// TIA Portal V19 export
FUNCTION "AUTO_SUBOUTPUT" : Void   // FC11, LAD
{ S7_Optimized_Access := 'TRUE' }
// stored: SetENOAutomatically false
BEGIN

REGION Network 1: MGF FEED PUMP P-101 A
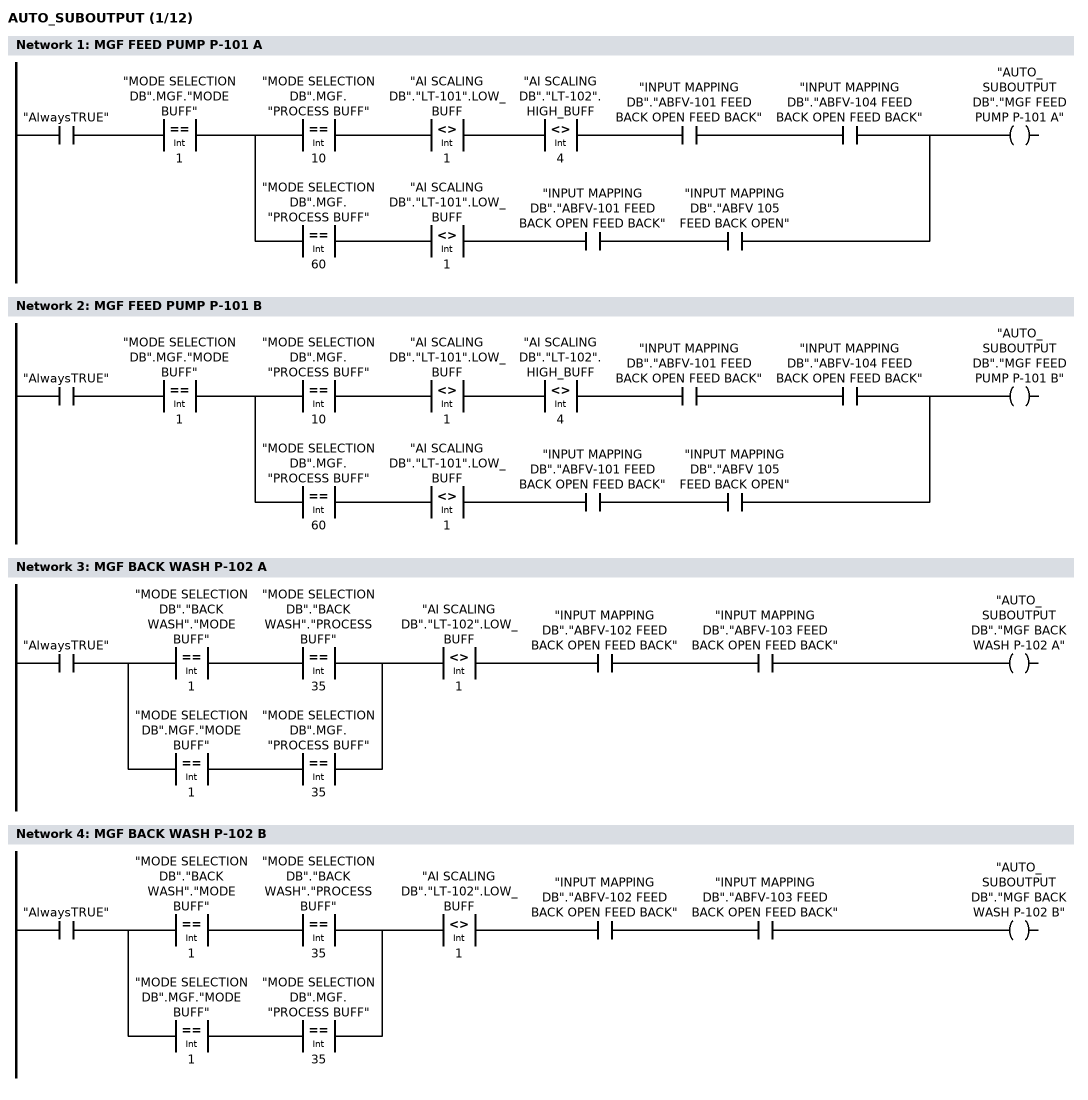
   RUNG wire#powerrail
      Contact( "AlwaysTRUE" )
      { S7_Templates := "SrcType := Int" } EQ_Contact(in1 := "MODE SELECTION DB".MGF."MODE BUFF", in2 := 1)
      wire#w1
      { S7_Templates := "SrcType := Int" } EQ_Contact(in1 := "MODE SELECTION DB".MGF."PROCESS BUFF", in2 := 10)
      { S7_Templates := "SrcType := Int" } NE_Contact(in1 := "AI SCALING DB"."LT-101".LOW_BUFF, in2 := 1)
      { S7_Templates := "SrcType := Int" } NE_Contact(in1 := "AI SCALING DB"."LT-102".HIGH_BUFF, in2 := 4)
      Contact( "INPUT MAPPING DB"."ABFV-101 FEED BACK OPEN FEED BACK" )
      Contact( "INPUT MAPPING DB"."ABFV-104 FEED BACK OPEN FEED BACK" )
      wire#w2
      Coil( "AUTO_SUBOUTPUT DB"."MGF FEED PUMP P-101 A" )
   END_RUNG
   RUNG wire#w1
      { S7_Templates := "SrcType := Int" } EQ_Contact(in1 := "MODE SELECTION DB".MGF."PROCESS BUFF", in2 := 60)
      { S7_Templates := "SrcType := Int" } NE_Contact(in1 := "AI SCALING DB"."LT-101".LOW_BUFF, in2 := 1)
      Contact( "INPUT MAPPING DB"."ABFV-101 FEED BACK OPEN FEED BACK" )
      Contact( "INPUT MAPPING DB"."ABFV 105 FEED BACK OPEN" )
   END_RUNG wire#w2
   // the same network as SCL:
   "AUTO_SUBOUTPUT DB"."MGF FEED PUMP P-101 A" := "AlwaysTRUE" AND ("MODE SELECTION DB".MGF."MODE BUFF" = 1) AND ((("MODE SELECTION DB".MGF."PROCESS BUFF" = 10) AND ("AI SCALING DB"."LT-101".LOW_BUFF <> 1) AND ("AI SCALING DB"."LT-102".HIGH_BUFF <> 4) AND "INPUT MAPPING DB"."ABFV-101 FEED BACK OPEN FEED BACK" AND "INPUT MAPPING DB"."ABFV-104 FEED BACK OPEN FEED BACK") OR (("MODE SELECTION DB".MGF."PROCESS BUFF" = 60) AND ("AI SCALING DB"."LT-101".LOW_BUFF <> 1) AND "INPUT MAPPING DB"."ABFV-101 FEED BACK OPEN FEED BACK" AND "INPUT MAPPING DB"."ABFV 105 FEED BACK OPEN"));
END_REGION

REGION Network 2: MGF FEED PUMP P-101 B
   RUNG wire#powerrail
      Contact( "AlwaysTRUE" )
      { S7_Templates := "SrcType := Int" } EQ_Contact(in1 := "MODE SELECTION DB".MGF."MODE BUFF", in2 := 1)
      wire#w1
      { S7_Templates := "SrcType := Int" } EQ_Contact(in1 := "MODE SELECTION DB".MGF."PROCESS BUFF", in2 := 10)
      { S7_Templates := "SrcType := Int" } NE_Contact(in1 := "AI SCALING DB"."LT-101".LOW_BUFF, in2 := 1)
      { S7_Templates := "SrcType := Int" } NE_Contact(in1 := "AI SCALING DB"."LT-102".HIGH_BUFF, in2 := 4)
      Contact( "INPUT MAPPING DB"."ABFV-101 FEED BACK OPEN FEED BACK" )
      Contact( "INPUT MAPPING DB"."ABFV-104 FEED BACK OPEN FEED BACK" )
      wire#w2
      Coil( "AUTO_SUBOUTPUT DB"."MGF FEED PUMP P-101 B" )
   END_RUNG
   RUNG wire#w1
      { S7_Templates := "SrcType := Int" } EQ_Contact(in1 := "MODE SELECTION DB".MGF."PROCESS BUFF", in2 := 60)
      { S7_Templates := "SrcType := Int" } NE_Contact(in1 := "AI SCALING DB"."LT-101".LOW_BUFF, in2 := 1)
      Contact( "INPUT MAPPING DB"."ABFV-101 FEED BACK OPEN FEED BACK" )
      Contact( "INPUT MAPPING DB"."ABFV 105 FEED BACK OPEN" )
   END_RUNG wire#w2
   // the same network as SCL:
   "AUTO_SUBOUTPUT DB"."MGF FEED PUMP P-101 B" := "AlwaysTRUE" AND ("MODE SELECTION DB".MGF."MODE BUFF" = 1) AND ((("MODE SELECTION DB".MGF."PROCESS BUFF" = 10) AND ("AI SCALING DB"."LT-101".LOW_BUFF <> 1) AND ("AI SCALING DB"."LT-102".HIGH_BUFF <> 4) AND "INPUT MAPPING DB"."ABFV-101 FEED BACK OPEN FEED BACK" AND "INPUT MAPPING DB"."ABFV-104 FEED BACK OPEN FEED BACK") OR (("MODE SELECTION DB".MGF."PROCESS BUFF" = 60) AND ("AI SCALING DB"."LT-101".LOW_BUFF <> 1) AND "INPUT MAPPING DB"."ABFV-101 FEED BACK OPEN FEED BACK" AND "INPUT MAPPING DB"."ABFV 105 FEED BACK OPEN"));
END_REGION

REGION Network 3: MGF BACK WASH P-102 A
   RUNG wire#powerrail
      Contact( "AlwaysTRUE" )
      wire#w1
      { S7_Templates := "SrcType := Int" } EQ_Contact(in1 := "MODE SELECTION DB"."BACK WASH"."MODE BUFF", in2 := 1)
      { S7_Templates := "SrcType := Int" } EQ_Contact(in1 := "MODE SELECTION DB"."BACK WASH"."PROCESS BUFF", in2 := 35)
      wire#w2
      { S7_Templates := "SrcType := Int" } NE_Contact(in1 := "AI SCALING DB"."LT-102".LOW_BUFF, in2 := 1)
      Contact( "INPUT MAPPING DB"."ABFV-102 FEED BACK OPEN FEED BACK" )
      Contact( "INPUT MAPPING DB"."ABFV-103 FEED BACK OPEN FEED BACK" )
      Coil( "AUTO_SUBOUTPUT DB"."MGF BACK WASH P-102 A" )
   END_RUNG
   RUNG wire#w1
      { S7_Templates := "SrcType := Int" } EQ_Contact(in1 := "MODE SELECTION DB".MGF."MODE BUFF", in2 := 1)
      { S7_Templates := "SrcType := Int" } EQ_Contact(in1 := "MODE SELECTION DB".MGF."PROCESS BUFF", in2 := 35)
   END_RUNG wire#w2
   // the same network as SCL:
   "AUTO_SUBOUTPUT DB"."MGF BACK WASH P-102 A" := "AlwaysTRUE" AND ((("MODE SELECTION DB"."BACK WASH"."MODE BUFF" = 1) AND ("MODE SELECTION DB"."BACK WASH"."PROCESS BUFF" = 35)) OR (("MODE SELECTION DB".MGF."MODE BUFF" = 1) AND ("MODE SELECTION DB".MGF."PROCESS BUFF" = 35))) AND ("AI SCALING DB"."LT-102".LOW_BUFF <> 1) AND "INPUT MAPPING DB"."ABFV-102 FEED BACK OPEN FEED BACK" AND "INPUT MAPPING DB"."ABFV-103 FEED BACK OPEN FEED BACK";
END_REGION

REGION Network 4: MGF BACK WASH P-102 B
   RUNG wire#powerrail
      Contact( "AlwaysTRUE" )
      wire#w1
      { S7_Templates := "SrcType := Int" } EQ_Contact(in1 := "MODE SELECTION DB"."BACK WASH"."MODE BUFF", in2 := 1)
      { S7_Templates := "SrcType := Int" } EQ_Contact(in1 := "MODE SELECTION DB"."BACK WASH"."PROCESS BUFF", in2 := 35)
      wire#w2
      { S7_Templates := "SrcType := Int" } NE_Contact(in1 := "AI SCALING DB"."LT-102".LOW_BUFF, in2 := 1)
      Contact( "INPUT MAPPING DB"."ABFV-102 FEED BACK OPEN FEED BACK" )
      Contact( "INPUT MAPPING DB"."ABFV-103 FEED BACK OPEN FEED BACK" )
      Coil( "AUTO_SUBOUTPUT DB"."MGF BACK WASH P-102 B" )
   END_RUNG
   RUNG wire#w1
      { S7_Templates := "SrcType := Int" } EQ_Contact(in1 := "MODE SELECTION DB".MGF."MODE BUFF", in2 := 1)
      { S7_Templates := "SrcType := Int" } EQ_Contact(in1 := "MODE SELECTION DB".MGF."PROCESS BUFF", in2 := 35)
   END_RUNG wire#w2
   // the same network as SCL:
   "AUTO_SUBOUTPUT DB"."MGF BACK WASH P-102 B" := "AlwaysTRUE" AND ((("MODE SELECTION DB"."BACK WASH"."MODE BUFF" = 1) AND ("MODE SELECTION DB"."BACK WASH"."PROCESS BUFF" = 35)) OR (("MODE SELECTION DB".MGF."MODE BUFF" = 1) AND ("MODE SELECTION DB".MGF."PROCESS BUFF" = 35))) AND ("AI SCALING DB"."LT-102".LOW_BUFF <> 1) AND "INPUT MAPPING DB"."ABFV-102 FEED BACK OPEN FEED BACK" AND "INPUT MAPPING DB"."ABFV-103 FEED BACK OPEN FEED BACK";
END_REGION

REGION Network 5: UF FEED PUMP P-103 A
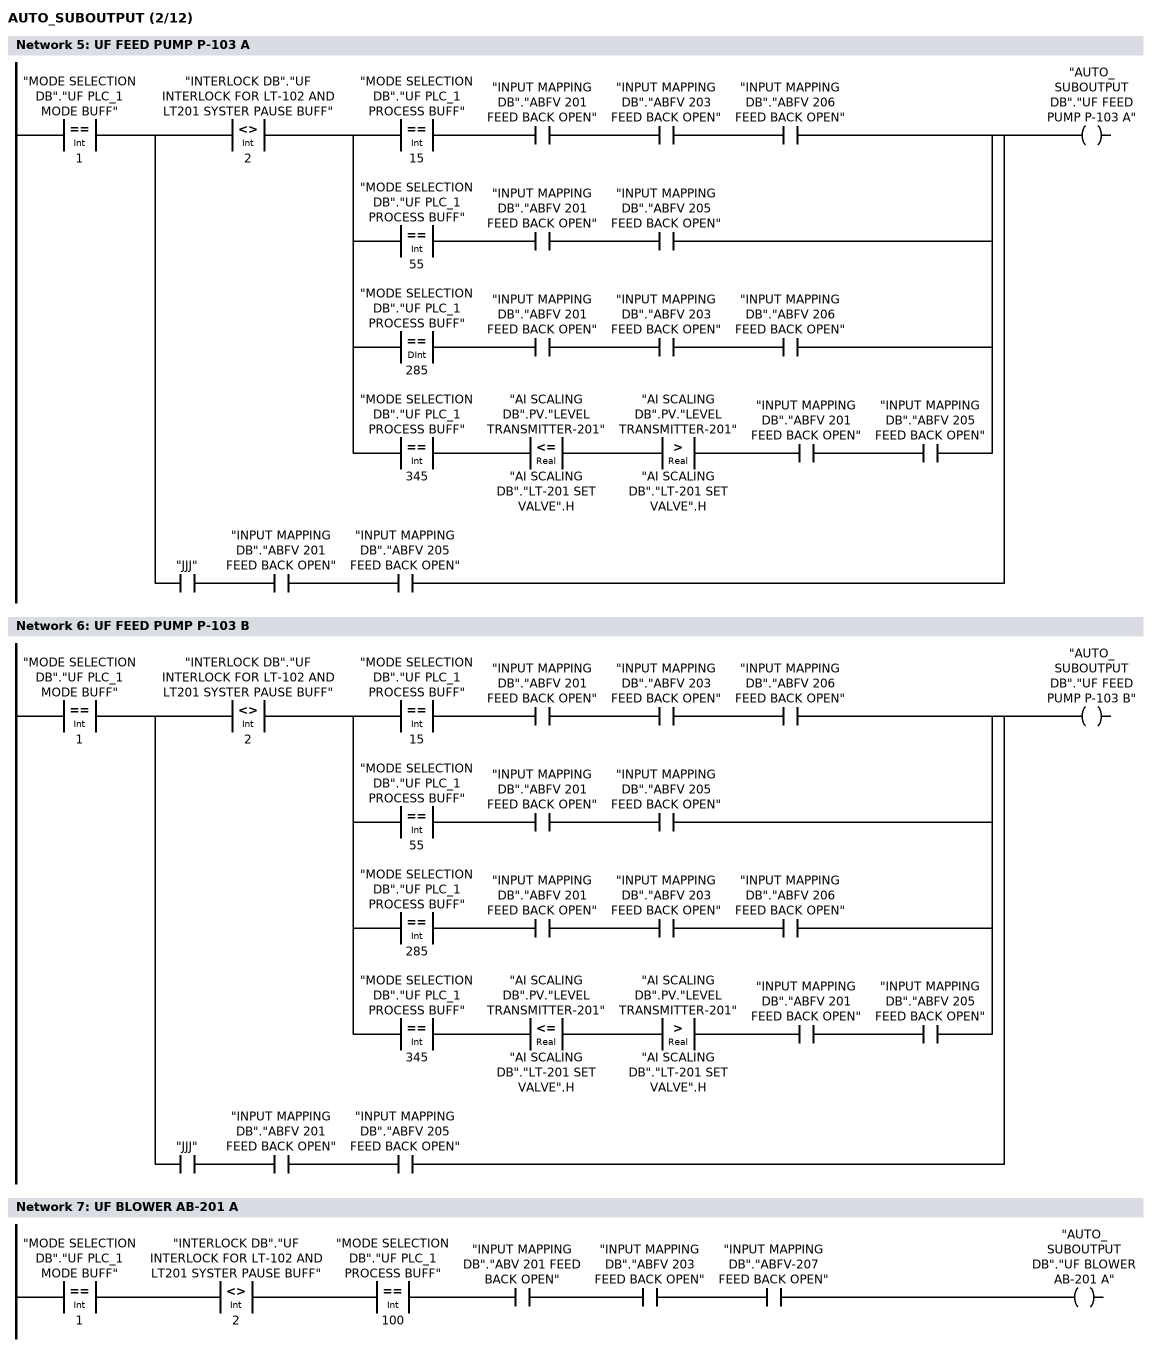
   RUNG wire#powerrail
      { S7_Templates := "SrcType := Int" } EQ_Contact(in1 := "MODE SELECTION DB"."UF PLC_1 MODE BUFF", in2 := 1)
      wire#w1
      { S7_Templates := "SrcType := Int" } NE_Contact(in1 := "INTERLOCK DB"."UF INTERLOCK FOR LT-102 AND LT201 SYSTER PAUSE BUFF", in2 := 2)
      wire#w2
      { S7_Templates := "SrcType := Int" } EQ_Contact(in1 := "MODE SELECTION DB"."UF PLC_1 PROCESS BUFF", in2 := 15)
      Contact( "INPUT MAPPING DB"."ABFV 201 FEED BACK OPEN" )
      Contact( "INPUT MAPPING DB"."ABFV 203 FEED BACK OPEN" )
      Contact( "INPUT MAPPING DB"."ABFV 206 FEED BACK OPEN" )
      wire#w3
      Coil( "AUTO_SUBOUTPUT DB"."UF FEED PUMP P-103 A" )
   END_RUNG
   RUNG wire#w2
      { S7_Templates := "SrcType := Int" } EQ_Contact(in1 := "MODE SELECTION DB"."UF PLC_1 PROCESS BUFF", in2 := 55)
      Contact( "INPUT MAPPING DB"."ABFV 201 FEED BACK OPEN" )
      Contact( "INPUT MAPPING DB"."ABFV 205 FEED BACK OPEN" )
   END_RUNG wire#w3
   RUNG wire#w2
      { S7_Templates := "SrcType := DInt" } EQ_Contact(in1 := "MODE SELECTION DB"."UF PLC_1 PROCESS BUFF", in2 := 285)
      Contact( "INPUT MAPPING DB"."ABFV 201 FEED BACK OPEN" )
      Contact( "INPUT MAPPING DB"."ABFV 203 FEED BACK OPEN" )
      Contact( "INPUT MAPPING DB"."ABFV 206 FEED BACK OPEN" )
   END_RUNG wire#w3
   RUNG wire#w2
      { S7_Templates := "SrcType := Int" } EQ_Contact(in1 := "MODE SELECTION DB"."UF PLC_1 PROCESS BUFF", in2 := 345)
      { S7_Templates := "SrcType := Real" } LE_Contact(in1 := "AI SCALING DB".PV."LEVEL TRANSMITTER-201", in2 := "AI SCALING DB"."LT-201 SET VALVE".H)
      { S7_Templates := "SrcType := Real" } GT_Contact(in1 := "AI SCALING DB".PV."LEVEL TRANSMITTER-201", in2 := "AI SCALING DB"."LT-201 SET VALVE".H)
      Contact( "INPUT MAPPING DB"."ABFV 201 FEED BACK OPEN" )
      Contact( "INPUT MAPPING DB"."ABFV 205 FEED BACK OPEN" )
   END_RUNG wire#w3
   RUNG wire#w1
      Contact( "JJJ" )
      Contact( "INPUT MAPPING DB"."ABFV 201 FEED BACK OPEN" )
      Contact( "INPUT MAPPING DB"."ABFV 205 FEED BACK OPEN" )
   END_RUNG wire#w3
   // the same network as SCL:
   "AUTO_SUBOUTPUT DB"."UF FEED PUMP P-103 A" := ("MODE SELECTION DB"."UF PLC_1 MODE BUFF" = 1) AND ((("INTERLOCK DB"."UF INTERLOCK FOR LT-102 AND LT201 SYSTER PAUSE BUFF" <> 2) AND ((("MODE SELECTION DB"."UF PLC_1 PROCESS BUFF" = 15) AND "INPUT MAPPING DB"."ABFV 201 FEED BACK OPEN" AND "INPUT MAPPING DB"."ABFV 203 FEED BACK OPEN" AND "INPUT MAPPING DB"."ABFV 206 FEED BACK OPEN") OR (("MODE SELECTION DB"."UF PLC_1 PROCESS BUFF" = 55) AND "INPUT MAPPING DB"."ABFV 201 FEED BACK OPEN" AND "INPUT MAPPING DB"."ABFV 205 FEED BACK OPEN") OR (("MODE SELECTION DB"."UF PLC_1 PROCESS BUFF" = 285) AND "INPUT MAPPING DB"."ABFV 201 FEED BACK OPEN" AND "INPUT MAPPING DB"."ABFV 203 FEED BACK OPEN" AND "INPUT MAPPING DB"."ABFV 206 FEED BACK OPEN") OR (("MODE SELECTION DB"."UF PLC_1 PROCESS BUFF" = 345) AND ("AI SCALING DB".PV."LEVEL TRANSMITTER-201" <= "AI SCALING DB"."LT-201 SET VALVE".H) AND ("AI SCALING DB".PV."LEVEL TRANSMITTER-201" > "AI SCALING DB"."LT-201 SET VALVE".H) AND "INPUT MAPPING DB"."ABFV 201 FEED BACK OPEN" AND "INPUT MAPPING DB"."ABFV 205 FEED BACK OPEN"))) OR ("JJJ" AND "INPUT MAPPING DB"."ABFV 201 FEED BACK OPEN" AND "INPUT MAPPING DB"."ABFV 205 FEED BACK OPEN"));
END_REGION

REGION Network 6: UF FEED PUMP P-103 B
   RUNG wire#powerrail
      { S7_Templates := "SrcType := Int" } EQ_Contact(in1 := "MODE SELECTION DB"."UF PLC_1 MODE BUFF", in2 := 1)
      wire#w1
      { S7_Templates := "SrcType := Int" } NE_Contact(in1 := "INTERLOCK DB"."UF INTERLOCK FOR LT-102 AND LT201 SYSTER PAUSE BUFF", in2 := 2)
      wire#w2
      { S7_Templates := "SrcType := Int" } EQ_Contact(in1 := "MODE SELECTION DB"."UF PLC_1 PROCESS BUFF", in2 := 15)
      Contact( "INPUT MAPPING DB"."ABFV 201 FEED BACK OPEN" )
      Contact( "INPUT MAPPING DB"."ABFV 203 FEED BACK OPEN" )
      Contact( "INPUT MAPPING DB"."ABFV 206 FEED BACK OPEN" )
      wire#w3
      Coil( "AUTO_SUBOUTPUT DB"."UF FEED PUMP P-103 B" )
   END_RUNG
   RUNG wire#w2
      { S7_Templates := "SrcType := Int" } EQ_Contact(in1 := "MODE SELECTION DB"."UF PLC_1 PROCESS BUFF", in2 := 55)
      Contact( "INPUT MAPPING DB"."ABFV 201 FEED BACK OPEN" )
      Contact( "INPUT MAPPING DB"."ABFV 205 FEED BACK OPEN" )
   END_RUNG wire#w3
   RUNG wire#w2
      { S7_Templates := "SrcType := Int" } EQ_Contact(in1 := "MODE SELECTION DB"."UF PLC_1 PROCESS BUFF", in2 := 285)
      Contact( "INPUT MAPPING DB"."ABFV 201 FEED BACK OPEN" )
      Contact( "INPUT MAPPING DB"."ABFV 203 FEED BACK OPEN" )
      Contact( "INPUT MAPPING DB"."ABFV 206 FEED BACK OPEN" )
   END_RUNG wire#w3
   RUNG wire#w2
      { S7_Templates := "SrcType := Int" } EQ_Contact(in1 := "MODE SELECTION DB"."UF PLC_1 PROCESS BUFF", in2 := 345)
      { S7_Templates := "SrcType := Real" } LE_Contact(in1 := "AI SCALING DB".PV."LEVEL TRANSMITTER-201", in2 := "AI SCALING DB"."LT-201 SET VALVE".H)
      { S7_Templates := "SrcType := Real" } GT_Contact(in1 := "AI SCALING DB".PV."LEVEL TRANSMITTER-201", in2 := "AI SCALING DB"."LT-201 SET VALVE".H)
      Contact( "INPUT MAPPING DB"."ABFV 201 FEED BACK OPEN" )
      Contact( "INPUT MAPPING DB"."ABFV 205 FEED BACK OPEN" )
   END_RUNG wire#w3
   RUNG wire#w1
      Contact( "JJJ" )
      Contact( "INPUT MAPPING DB"."ABFV 201 FEED BACK OPEN" )
      Contact( "INPUT MAPPING DB"."ABFV 205 FEED BACK OPEN" )
   END_RUNG wire#w3
   // the same network as SCL:
   "AUTO_SUBOUTPUT DB"."UF FEED PUMP P-103 B" := ("MODE SELECTION DB"."UF PLC_1 MODE BUFF" = 1) AND ((("INTERLOCK DB"."UF INTERLOCK FOR LT-102 AND LT201 SYSTER PAUSE BUFF" <> 2) AND ((("MODE SELECTION DB"."UF PLC_1 PROCESS BUFF" = 15) AND "INPUT MAPPING DB"."ABFV 201 FEED BACK OPEN" AND "INPUT MAPPING DB"."ABFV 203 FEED BACK OPEN" AND "INPUT MAPPING DB"."ABFV 206 FEED BACK OPEN") OR (("MODE SELECTION DB"."UF PLC_1 PROCESS BUFF" = 55) AND "INPUT MAPPING DB"."ABFV 201 FEED BACK OPEN" AND "INPUT MAPPING DB"."ABFV 205 FEED BACK OPEN") OR (("MODE SELECTION DB"."UF PLC_1 PROCESS BUFF" = 285) AND "INPUT MAPPING DB"."ABFV 201 FEED BACK OPEN" AND "INPUT MAPPING DB"."ABFV 203 FEED BACK OPEN" AND "INPUT MAPPING DB"."ABFV 206 FEED BACK OPEN") OR (("MODE SELECTION DB"."UF PLC_1 PROCESS BUFF" = 345) AND ("AI SCALING DB".PV."LEVEL TRANSMITTER-201" <= "AI SCALING DB"."LT-201 SET VALVE".H) AND ("AI SCALING DB".PV."LEVEL TRANSMITTER-201" > "AI SCALING DB"."LT-201 SET VALVE".H) AND "INPUT MAPPING DB"."ABFV 201 FEED BACK OPEN" AND "INPUT MAPPING DB"."ABFV 205 FEED BACK OPEN"))) OR ("JJJ" AND "INPUT MAPPING DB"."ABFV 201 FEED BACK OPEN" AND "INPUT MAPPING DB"."ABFV 205 FEED BACK OPEN"));
END_REGION

REGION Network 7: UF BLOWER AB-201 A
   RUNG wire#powerrail
      { S7_Templates := "SrcType := Int" } EQ_Contact(in1 := "MODE SELECTION DB"."UF PLC_1 MODE BUFF", in2 := 1)
      { S7_Templates := "SrcType := Int" } NE_Contact(in1 := "INTERLOCK DB"."UF INTERLOCK FOR LT-102 AND LT201 SYSTER PAUSE BUFF", in2 := 2)
      { S7_Templates := "SrcType := Int" } EQ_Contact(in1 := "MODE SELECTION DB"."UF PLC_1 PROCESS BUFF", in2 := 100)
      Contact( "INPUT MAPPING DB"."ABV 201 FEED BACK OPEN" )
      Contact( "INPUT MAPPING DB"."ABFV 203 FEED BACK OPEN" )
      Contact( "INPUT MAPPING DB"."ABFV-207 FEED BACK OPEN" )
      Coil( "AUTO_SUBOUTPUT DB"."UF BLOWER AB-201 A" )
   END_RUNG
   // the same network as SCL:
   "AUTO_SUBOUTPUT DB"."UF BLOWER AB-201 A" := ("MODE SELECTION DB"."UF PLC_1 MODE BUFF" = 1) AND ("INTERLOCK DB"."UF INTERLOCK FOR LT-102 AND LT201 SYSTER PAUSE BUFF" <> 2) AND ("MODE SELECTION DB"."UF PLC_1 PROCESS BUFF" = 100) AND "INPUT MAPPING DB"."ABV 201 FEED BACK OPEN" AND "INPUT MAPPING DB"."ABFV 203 FEED BACK OPEN" AND "INPUT MAPPING DB"."ABFV-207 FEED BACK OPEN";
END_REGION

REGION Network 8: UF BLOWER AB 201 B
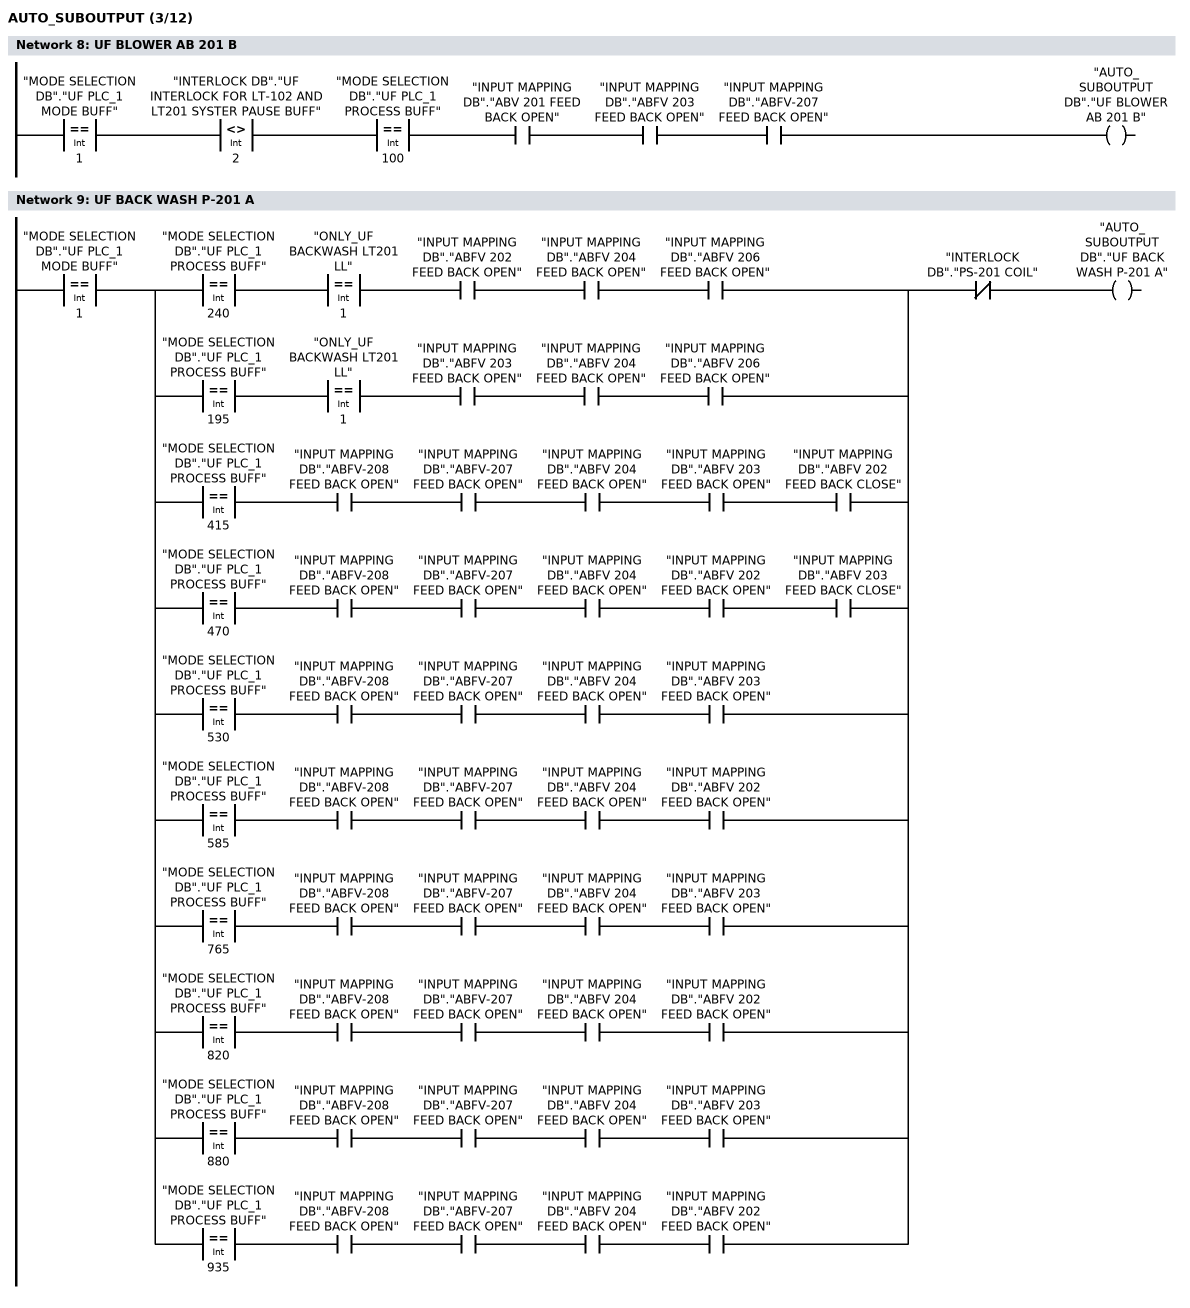
   RUNG wire#powerrail
      { S7_Templates := "SrcType := Int" } EQ_Contact(in1 := "MODE SELECTION DB"."UF PLC_1 MODE BUFF", in2 := 1)
      { S7_Templates := "SrcType := Int" } NE_Contact(in1 := "INTERLOCK DB"."UF INTERLOCK FOR LT-102 AND LT201 SYSTER PAUSE BUFF", in2 := 2)
      { S7_Templates := "SrcType := Int" } EQ_Contact(in1 := "MODE SELECTION DB"."UF PLC_1 PROCESS BUFF", in2 := 100)
      Contact( "INPUT MAPPING DB"."ABV 201 FEED BACK OPEN" )
      Contact( "INPUT MAPPING DB"."ABFV 203 FEED BACK OPEN" )
      Contact( "INPUT MAPPING DB"."ABFV-207 FEED BACK OPEN" )
      Coil( "AUTO_SUBOUTPUT DB"."UF BLOWER AB 201 B" )
   END_RUNG
   // the same network as SCL:
   "AUTO_SUBOUTPUT DB"."UF BLOWER AB 201 B" := ("MODE SELECTION DB"."UF PLC_1 MODE BUFF" = 1) AND ("INTERLOCK DB"."UF INTERLOCK FOR LT-102 AND LT201 SYSTER PAUSE BUFF" <> 2) AND ("MODE SELECTION DB"."UF PLC_1 PROCESS BUFF" = 100) AND "INPUT MAPPING DB"."ABV 201 FEED BACK OPEN" AND "INPUT MAPPING DB"."ABFV 203 FEED BACK OPEN" AND "INPUT MAPPING DB"."ABFV-207 FEED BACK OPEN";
END_REGION

REGION Network 9: UF BACK WASH P-201 A
   RUNG wire#powerrail
      { S7_Templates := "SrcType := Int" } EQ_Contact(in1 := "MODE SELECTION DB"."UF PLC_1 MODE BUFF", in2 := 1)
      wire#w1
      { S7_Templates := "SrcType := Int" } EQ_Contact(in1 := "MODE SELECTION DB"."UF PLC_1 PROCESS BUFF", in2 := 240)
      { S7_Templates := "SrcType := Int" } EQ_Contact(in1 := "ONLY_UF BACKWASH LT201 LL", in2 := 1)
      Contact( "INPUT MAPPING DB"."ABFV 202 FEED BACK OPEN" )
      Contact( "INPUT MAPPING DB"."ABFV 204 FEED BACK OPEN" )
      Contact( "INPUT MAPPING DB"."ABFV 206 FEED BACK OPEN" )
      wire#w2
      I_Contact( "INTERLOCK DB"."PS-201 COIL" )
      Coil( "AUTO_SUBOUTPUT DB"."UF BACK WASH P-201 A" )
   END_RUNG
   RUNG wire#w1
      { S7_Templates := "SrcType := Int" } EQ_Contact(in1 := "MODE SELECTION DB"."UF PLC_1 PROCESS BUFF", in2 := 195)
      { S7_Templates := "SrcType := Int" } EQ_Contact(in1 := "ONLY_UF BACKWASH LT201 LL", in2 := 1)
      Contact( "INPUT MAPPING DB"."ABFV 203 FEED BACK OPEN" )
      Contact( "INPUT MAPPING DB"."ABFV 204 FEED BACK OPEN" )
      Contact( "INPUT MAPPING DB"."ABFV 206 FEED BACK OPEN" )
   END_RUNG wire#w2
   RUNG wire#w1
      { S7_Templates := "SrcType := Int" } EQ_Contact(in1 := "MODE SELECTION DB"."UF PLC_1 PROCESS BUFF", in2 := 415)
      Contact( "INPUT MAPPING DB"."ABFV-208 FEED BACK OPEN" )
      Contact( "INPUT MAPPING DB"."ABFV-207 FEED BACK OPEN" )
      Contact( "INPUT MAPPING DB"."ABFV 204 FEED BACK OPEN" )
      Contact( "INPUT MAPPING DB"."ABFV 203 FEED BACK OPEN" )
      Contact( "INPUT MAPPING DB"."ABFV 202 FEED BACK CLOSE" )
   END_RUNG wire#w2
   RUNG wire#w1
      { S7_Templates := "SrcType := Int" } EQ_Contact(in1 := "MODE SELECTION DB"."UF PLC_1 PROCESS BUFF", in2 := 470)
      Contact( "INPUT MAPPING DB"."ABFV-208 FEED BACK OPEN" )
      Contact( "INPUT MAPPING DB"."ABFV-207 FEED BACK OPEN" )
      Contact( "INPUT MAPPING DB"."ABFV 204 FEED BACK OPEN" )
      Contact( "INPUT MAPPING DB"."ABFV 202 FEED BACK OPEN" )
      Contact( "INPUT MAPPING DB"."ABFV 203 FEED BACK CLOSE" )
   END_RUNG wire#w2
   RUNG wire#w1
      { S7_Templates := "SrcType := Int" } EQ_Contact(in1 := "MODE SELECTION DB"."UF PLC_1 PROCESS BUFF", in2 := 530)
      Contact( "INPUT MAPPING DB"."ABFV-208 FEED BACK OPEN" )
      Contact( "INPUT MAPPING DB"."ABFV-207 FEED BACK OPEN" )
      Contact( "INPUT MAPPING DB"."ABFV 204 FEED BACK OPEN" )
      Contact( "INPUT MAPPING DB"."ABFV 203 FEED BACK OPEN" )
   END_RUNG wire#w2
   RUNG wire#w1
      { S7_Templates := "SrcType := Int" } EQ_Contact(in1 := "MODE SELECTION DB"."UF PLC_1 PROCESS BUFF", in2 := 585)
      Contact( "INPUT MAPPING DB"."ABFV-208 FEED BACK OPEN" )
      Contact( "INPUT MAPPING DB"."ABFV-207 FEED BACK OPEN" )
      Contact( "INPUT MAPPING DB"."ABFV 204 FEED BACK OPEN" )
      Contact( "INPUT MAPPING DB"."ABFV 202 FEED BACK OPEN" )
   END_RUNG wire#w2
   RUNG wire#w1
      { S7_Templates := "SrcType := Int" } EQ_Contact(in1 := "MODE SELECTION DB"."UF PLC_1 PROCESS BUFF", in2 := 765)
      Contact( "INPUT MAPPING DB"."ABFV-208 FEED BACK OPEN" )
      Contact( "INPUT MAPPING DB"."ABFV-207 FEED BACK OPEN" )
      Contact( "INPUT MAPPING DB"."ABFV 204 FEED BACK OPEN" )
      Contact( "INPUT MAPPING DB"."ABFV 203 FEED BACK OPEN" )
   END_RUNG wire#w2
   RUNG wire#w1
      { S7_Templates := "SrcType := Int" } EQ_Contact(in1 := "MODE SELECTION DB"."UF PLC_1 PROCESS BUFF", in2 := 820)
      Contact( "INPUT MAPPING DB"."ABFV-208 FEED BACK OPEN" )
      Contact( "INPUT MAPPING DB"."ABFV-207 FEED BACK OPEN" )
      Contact( "INPUT MAPPING DB"."ABFV 204 FEED BACK OPEN" )
      Contact( "INPUT MAPPING DB"."ABFV 202 FEED BACK OPEN" )
   END_RUNG wire#w2
   RUNG wire#w1
      { S7_Templates := "SrcType := Int" } EQ_Contact(in1 := "MODE SELECTION DB"."UF PLC_1 PROCESS BUFF", in2 := 880)
      Contact( "INPUT MAPPING DB"."ABFV-208 FEED BACK OPEN" )
      Contact( "INPUT MAPPING DB"."ABFV-207 FEED BACK OPEN" )
      Contact( "INPUT MAPPING DB"."ABFV 204 FEED BACK OPEN" )
      Contact( "INPUT MAPPING DB"."ABFV 203 FEED BACK OPEN" )
   END_RUNG wire#w2
   RUNG wire#w1
      { S7_Templates := "SrcType := Int" } EQ_Contact(in1 := "MODE SELECTION DB"."UF PLC_1 PROCESS BUFF", in2 := 935)
      Contact( "INPUT MAPPING DB"."ABFV-208 FEED BACK OPEN" )
      Contact( "INPUT MAPPING DB"."ABFV-207 FEED BACK OPEN" )
      Contact( "INPUT MAPPING DB"."ABFV 204 FEED BACK OPEN" )
      Contact( "INPUT MAPPING DB"."ABFV 202 FEED BACK OPEN" )
   END_RUNG wire#w2
   // the same network as SCL:
   "AUTO_SUBOUTPUT DB"."UF BACK WASH P-201 A" := ("MODE SELECTION DB"."UF PLC_1 MODE BUFF" = 1) AND ((("MODE SELECTION DB"."UF PLC_1 PROCESS BUFF" = 240) AND ("ONLY_UF BACKWASH LT201 LL" = 1) AND "INPUT MAPPING DB"."ABFV 202 FEED BACK OPEN" AND "INPUT MAPPING DB"."ABFV 204 FEED BACK OPEN" AND "INPUT MAPPING DB"."ABFV 206 FEED BACK OPEN") OR (("MODE SELECTION DB"."UF PLC_1 PROCESS BUFF" = 195) AND ("ONLY_UF BACKWASH LT201 LL" = 1) AND "INPUT MAPPING DB"."ABFV 203 FEED BACK OPEN" AND "INPUT MAPPING DB"."ABFV 204 FEED BACK OPEN" AND "INPUT MAPPING DB"."ABFV 206 FEED BACK OPEN") OR (("MODE SELECTION DB"."UF PLC_1 PROCESS BUFF" = 415) AND "INPUT MAPPING DB"."ABFV-208 FEED BACK OPEN" AND "INPUT MAPPING DB"."ABFV-207 FEED BACK OPEN" AND "INPUT MAPPING DB"."ABFV 204 FEED BACK OPEN" AND "INPUT MAPPING DB"."ABFV 203 FEED BACK OPEN" AND "INPUT MAPPING DB"."ABFV 202 FEED BACK CLOSE") OR (("MODE SELECTION DB"."UF PLC_1 PROCESS BUFF" = 470) AND "INPUT MAPPING DB"."ABFV-208 FEED BACK OPEN" AND "INPUT MAPPING DB"."ABFV-207 FEED BACK OPEN" AND "INPUT MAPPING DB"."ABFV 204 FEED BACK OPEN" AND "INPUT MAPPING DB"."ABFV 202 FEED BACK OPEN" AND "INPUT MAPPING DB"."ABFV 203 FEED BACK CLOSE") OR (("MODE SELECTION DB"."UF PLC_1 PROCESS BUFF" = 530) AND "INPUT MAPPING DB"."ABFV-208 FEED BACK OPEN" AND "INPUT MAPPING DB"."ABFV-207 FEED BACK OPEN" AND "INPUT MAPPING DB"."ABFV 204 FEED BACK OPEN" AND "INPUT MAPPING DB"."ABFV 203 FEED BACK OPEN") OR (("MODE SELECTION DB"."UF PLC_1 PROCESS BUFF" = 585) AND "INPUT MAPPING DB"."ABFV-208 FEED BACK OPEN" AND "INPUT MAPPING DB"."ABFV-207 FEED BACK OPEN" AND "INPUT MAPPING DB"."ABFV 204 FEED BACK OPEN" AND "INPUT MAPPING DB"."ABFV 202 FEED BACK OPEN") OR (("MODE SELECTION DB"."UF PLC_1 PROCESS BUFF" = 765) AND "INPUT MAPPING DB"."ABFV-208 FEED BACK OPEN" AND "INPUT MAPPING DB"."ABFV-207 FEED BACK OPEN" AND "INPUT MAPPING DB"."ABFV 204 FEED BACK OPEN" AND "INPUT MAPPING DB"."ABFV 203 FEED BACK OPEN") OR (("MODE SELECTION DB"."UF PLC_1 PROCESS BUFF" = 820) AND "INPUT MAPPING DB"."ABFV-208 FEED BACK OPEN" AND "INPUT MAPPING DB"."ABFV-207 FEED BACK OPEN" AND "INPUT MAPPING DB"."ABFV 204 FEED BACK OPEN" AND "INPUT MAPPING DB"."ABFV 202 FEED BACK OPEN") OR (("MODE SELECTION DB"."UF PLC_1 PROCESS BUFF" = 880) AND "INPUT MAPPING DB"."ABFV-208 FEED BACK OPEN" AND "INPUT MAPPING DB"."ABFV-207 FEED BACK OPEN" AND "INPUT MAPPING DB"."ABFV 204 FEED BACK OPEN" AND "INPUT MAPPING DB"."ABFV 203 FEED BACK OPEN") OR (("MODE SELECTION DB"."UF PLC_1 PROCESS BUFF" = 935) AND "INPUT MAPPING DB"."ABFV-208 FEED BACK OPEN" AND "INPUT MAPPING DB"."ABFV-207 FEED BACK OPEN" AND "INPUT MAPPING DB"."ABFV 204 FEED BACK OPEN" AND "INPUT MAPPING DB"."ABFV 202 FEED BACK OPEN")) AND NOT "INTERLOCK DB"."PS-201 COIL";
END_REGION

REGION Network 10: UF BACK WASH P-201 B
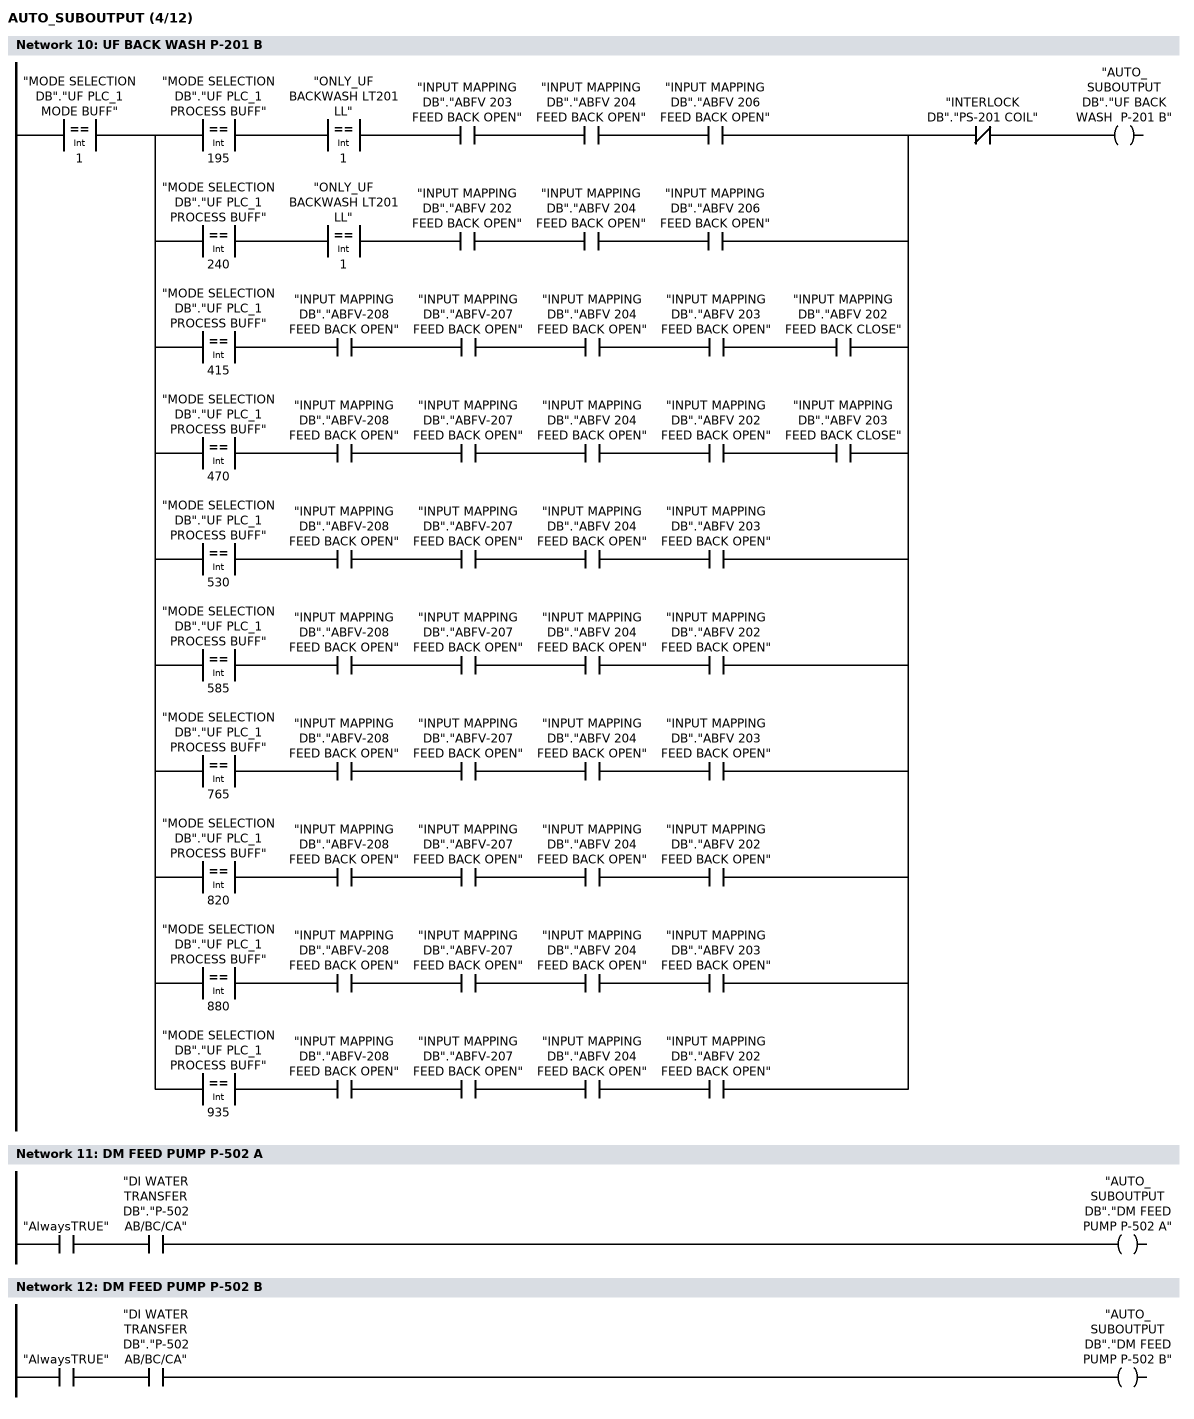
   RUNG wire#powerrail
      { S7_Templates := "SrcType := Int" } EQ_Contact(in1 := "MODE SELECTION DB"."UF PLC_1 MODE BUFF", in2 := 1)
      wire#w1
      { S7_Templates := "SrcType := Int" } EQ_Contact(in1 := "MODE SELECTION DB"."UF PLC_1 PROCESS BUFF", in2 := 195)
      { S7_Templates := "SrcType := Int" } EQ_Contact(in1 := "ONLY_UF BACKWASH LT201 LL", in2 := 1)
      Contact( "INPUT MAPPING DB"."ABFV 203 FEED BACK OPEN" )
      Contact( "INPUT MAPPING DB"."ABFV 204 FEED BACK OPEN" )
      Contact( "INPUT MAPPING DB"."ABFV 206 FEED BACK OPEN" )
      wire#w2
      I_Contact( "INTERLOCK DB"."PS-201 COIL" )
      Coil( "AUTO_SUBOUTPUT DB"."UF BACK WASH  P-201 B" )
   END_RUNG
   RUNG wire#w1
      { S7_Templates := "SrcType := Int" } EQ_Contact(in1 := "MODE SELECTION DB"."UF PLC_1 PROCESS BUFF", in2 := 240)
      { S7_Templates := "SrcType := Int" } EQ_Contact(in1 := "ONLY_UF BACKWASH LT201 LL", in2 := 1)
      Contact( "INPUT MAPPING DB"."ABFV 202 FEED BACK OPEN" )
      Contact( "INPUT MAPPING DB"."ABFV 204 FEED BACK OPEN" )
      Contact( "INPUT MAPPING DB"."ABFV 206 FEED BACK OPEN" )
   END_RUNG wire#w2
   RUNG wire#w1
      { S7_Templates := "SrcType := Int" } EQ_Contact(in1 := "MODE SELECTION DB"."UF PLC_1 PROCESS BUFF", in2 := 415)
      Contact( "INPUT MAPPING DB"."ABFV-208 FEED BACK OPEN" )
      Contact( "INPUT MAPPING DB"."ABFV-207 FEED BACK OPEN" )
      Contact( "INPUT MAPPING DB"."ABFV 204 FEED BACK OPEN" )
      Contact( "INPUT MAPPING DB"."ABFV 203 FEED BACK OPEN" )
      Contact( "INPUT MAPPING DB"."ABFV 202 FEED BACK CLOSE" )
   END_RUNG wire#w2
   RUNG wire#w1
      { S7_Templates := "SrcType := Int" } EQ_Contact(in1 := "MODE SELECTION DB"."UF PLC_1 PROCESS BUFF", in2 := 470)
      Contact( "INPUT MAPPING DB"."ABFV-208 FEED BACK OPEN" )
      Contact( "INPUT MAPPING DB"."ABFV-207 FEED BACK OPEN" )
      Contact( "INPUT MAPPING DB"."ABFV 204 FEED BACK OPEN" )
      Contact( "INPUT MAPPING DB"."ABFV 202 FEED BACK OPEN" )
      Contact( "INPUT MAPPING DB"."ABFV 203 FEED BACK CLOSE" )
   END_RUNG wire#w2
   RUNG wire#w1
      { S7_Templates := "SrcType := Int" } EQ_Contact(in1 := "MODE SELECTION DB"."UF PLC_1 PROCESS BUFF", in2 := 530)
      Contact( "INPUT MAPPING DB"."ABFV-208 FEED BACK OPEN" )
      Contact( "INPUT MAPPING DB"."ABFV-207 FEED BACK OPEN" )
      Contact( "INPUT MAPPING DB"."ABFV 204 FEED BACK OPEN" )
      Contact( "INPUT MAPPING DB"."ABFV 203 FEED BACK OPEN" )
   END_RUNG wire#w2
   RUNG wire#w1
      { S7_Templates := "SrcType := Int" } EQ_Contact(in1 := "MODE SELECTION DB"."UF PLC_1 PROCESS BUFF", in2 := 585)
      Contact( "INPUT MAPPING DB"."ABFV-208 FEED BACK OPEN" )
      Contact( "INPUT MAPPING DB"."ABFV-207 FEED BACK OPEN" )
      Contact( "INPUT MAPPING DB"."ABFV 204 FEED BACK OPEN" )
      Contact( "INPUT MAPPING DB"."ABFV 202 FEED BACK OPEN" )
   END_RUNG wire#w2
   RUNG wire#w1
      { S7_Templates := "SrcType := Int" } EQ_Contact(in1 := "MODE SELECTION DB"."UF PLC_1 PROCESS BUFF", in2 := 765)
      Contact( "INPUT MAPPING DB"."ABFV-208 FEED BACK OPEN" )
      Contact( "INPUT MAPPING DB"."ABFV-207 FEED BACK OPEN" )
      Contact( "INPUT MAPPING DB"."ABFV 204 FEED BACK OPEN" )
      Contact( "INPUT MAPPING DB"."ABFV 203 FEED BACK OPEN" )
   END_RUNG wire#w2
   RUNG wire#w1
      { S7_Templates := "SrcType := Int" } EQ_Contact(in1 := "MODE SELECTION DB"."UF PLC_1 PROCESS BUFF", in2 := 820)
      Contact( "INPUT MAPPING DB"."ABFV-208 FEED BACK OPEN" )
      Contact( "INPUT MAPPING DB"."ABFV-207 FEED BACK OPEN" )
      Contact( "INPUT MAPPING DB"."ABFV 204 FEED BACK OPEN" )
      Contact( "INPUT MAPPING DB"."ABFV 202 FEED BACK OPEN" )
   END_RUNG wire#w2
   RUNG wire#w1
      { S7_Templates := "SrcType := Int" } EQ_Contact(in1 := "MODE SELECTION DB"."UF PLC_1 PROCESS BUFF", in2 := 880)
      Contact( "INPUT MAPPING DB"."ABFV-208 FEED BACK OPEN" )
      Contact( "INPUT MAPPING DB"."ABFV-207 FEED BACK OPEN" )
      Contact( "INPUT MAPPING DB"."ABFV 204 FEED BACK OPEN" )
      Contact( "INPUT MAPPING DB"."ABFV 203 FEED BACK OPEN" )
   END_RUNG wire#w2
   RUNG wire#w1
      { S7_Templates := "SrcType := Int" } EQ_Contact(in1 := "MODE SELECTION DB"."UF PLC_1 PROCESS BUFF", in2 := 935)
      Contact( "INPUT MAPPING DB"."ABFV-208 FEED BACK OPEN" )
      Contact( "INPUT MAPPING DB"."ABFV-207 FEED BACK OPEN" )
      Contact( "INPUT MAPPING DB"."ABFV 204 FEED BACK OPEN" )
      Contact( "INPUT MAPPING DB"."ABFV 202 FEED BACK OPEN" )
   END_RUNG wire#w2
   // the same network as SCL:
   "AUTO_SUBOUTPUT DB"."UF BACK WASH  P-201 B" := ("MODE SELECTION DB"."UF PLC_1 MODE BUFF" = 1) AND ((("MODE SELECTION DB"."UF PLC_1 PROCESS BUFF" = 195) AND ("ONLY_UF BACKWASH LT201 LL" = 1) AND "INPUT MAPPING DB"."ABFV 203 FEED BACK OPEN" AND "INPUT MAPPING DB"."ABFV 204 FEED BACK OPEN" AND "INPUT MAPPING DB"."ABFV 206 FEED BACK OPEN") OR (("MODE SELECTION DB"."UF PLC_1 PROCESS BUFF" = 240) AND ("ONLY_UF BACKWASH LT201 LL" = 1) AND "INPUT MAPPING DB"."ABFV 202 FEED BACK OPEN" AND "INPUT MAPPING DB"."ABFV 204 FEED BACK OPEN" AND "INPUT MAPPING DB"."ABFV 206 FEED BACK OPEN") OR (("MODE SELECTION DB"."UF PLC_1 PROCESS BUFF" = 415) AND "INPUT MAPPING DB"."ABFV-208 FEED BACK OPEN" AND "INPUT MAPPING DB"."ABFV-207 FEED BACK OPEN" AND "INPUT MAPPING DB"."ABFV 204 FEED BACK OPEN" AND "INPUT MAPPING DB"."ABFV 203 FEED BACK OPEN" AND "INPUT MAPPING DB"."ABFV 202 FEED BACK CLOSE") OR (("MODE SELECTION DB"."UF PLC_1 PROCESS BUFF" = 470) AND "INPUT MAPPING DB"."ABFV-208 FEED BACK OPEN" AND "INPUT MAPPING DB"."ABFV-207 FEED BACK OPEN" AND "INPUT MAPPING DB"."ABFV 204 FEED BACK OPEN" AND "INPUT MAPPING DB"."ABFV 202 FEED BACK OPEN" AND "INPUT MAPPING DB"."ABFV 203 FEED BACK CLOSE") OR (("MODE SELECTION DB"."UF PLC_1 PROCESS BUFF" = 530) AND "INPUT MAPPING DB"."ABFV-208 FEED BACK OPEN" AND "INPUT MAPPING DB"."ABFV-207 FEED BACK OPEN" AND "INPUT MAPPING DB"."ABFV 204 FEED BACK OPEN" AND "INPUT MAPPING DB"."ABFV 203 FEED BACK OPEN") OR (("MODE SELECTION DB"."UF PLC_1 PROCESS BUFF" = 585) AND "INPUT MAPPING DB"."ABFV-208 FEED BACK OPEN" AND "INPUT MAPPING DB"."ABFV-207 FEED BACK OPEN" AND "INPUT MAPPING DB"."ABFV 204 FEED BACK OPEN" AND "INPUT MAPPING DB"."ABFV 202 FEED BACK OPEN") OR (("MODE SELECTION DB"."UF PLC_1 PROCESS BUFF" = 765) AND "INPUT MAPPING DB"."ABFV-208 FEED BACK OPEN" AND "INPUT MAPPING DB"."ABFV-207 FEED BACK OPEN" AND "INPUT MAPPING DB"."ABFV 204 FEED BACK OPEN" AND "INPUT MAPPING DB"."ABFV 203 FEED BACK OPEN") OR (("MODE SELECTION DB"."UF PLC_1 PROCESS BUFF" = 820) AND "INPUT MAPPING DB"."ABFV-208 FEED BACK OPEN" AND "INPUT MAPPING DB"."ABFV-207 FEED BACK OPEN" AND "INPUT MAPPING DB"."ABFV 204 FEED BACK OPEN" AND "INPUT MAPPING DB"."ABFV 202 FEED BACK OPEN") OR (("MODE SELECTION DB"."UF PLC_1 PROCESS BUFF" = 880) AND "INPUT MAPPING DB"."ABFV-208 FEED BACK OPEN" AND "INPUT MAPPING DB"."ABFV-207 FEED BACK OPEN" AND "INPUT MAPPING DB"."ABFV 204 FEED BACK OPEN" AND "INPUT MAPPING DB"."ABFV 203 FEED BACK OPEN") OR (("MODE SELECTION DB"."UF PLC_1 PROCESS BUFF" = 935) AND "INPUT MAPPING DB"."ABFV-208 FEED BACK OPEN" AND "INPUT MAPPING DB"."ABFV-207 FEED BACK OPEN" AND "INPUT MAPPING DB"."ABFV 204 FEED BACK OPEN" AND "INPUT MAPPING DB"."ABFV 202 FEED BACK OPEN")) AND NOT "INTERLOCK DB"."PS-201 COIL";
END_REGION

REGION Network 11: DM FEED PUMP P-502 A
   RUNG wire#powerrail
      Contact( "AlwaysTRUE" )
      Contact( "DI WATER TRANSFER DB"."P-502 AB/BC/CA" )
      Coil( "AUTO_SUBOUTPUT DB"."DM FEED PUMP P-502 A" )
   END_RUNG
   // the same network as SCL:
   "AUTO_SUBOUTPUT DB"."DM FEED PUMP P-502 A" := "AlwaysTRUE" AND "DI WATER TRANSFER DB"."P-502 AB/BC/CA";
END_REGION

REGION Network 12: DM FEED PUMP P-502 B
   RUNG wire#powerrail
      Contact( "AlwaysTRUE" )
      Contact( "DI WATER TRANSFER DB"."P-502 AB/BC/CA" )
      Coil( "AUTO_SUBOUTPUT DB"."DM FEED PUMP P-502 B" )
   END_RUNG
   // the same network as SCL:
   "AUTO_SUBOUTPUT DB"."DM FEED PUMP P-502 B" := "AlwaysTRUE" AND "DI WATER TRANSFER DB"."P-502 AB/BC/CA";
END_REGION

REGION Network 13: DM FEED PUMP P-502 C
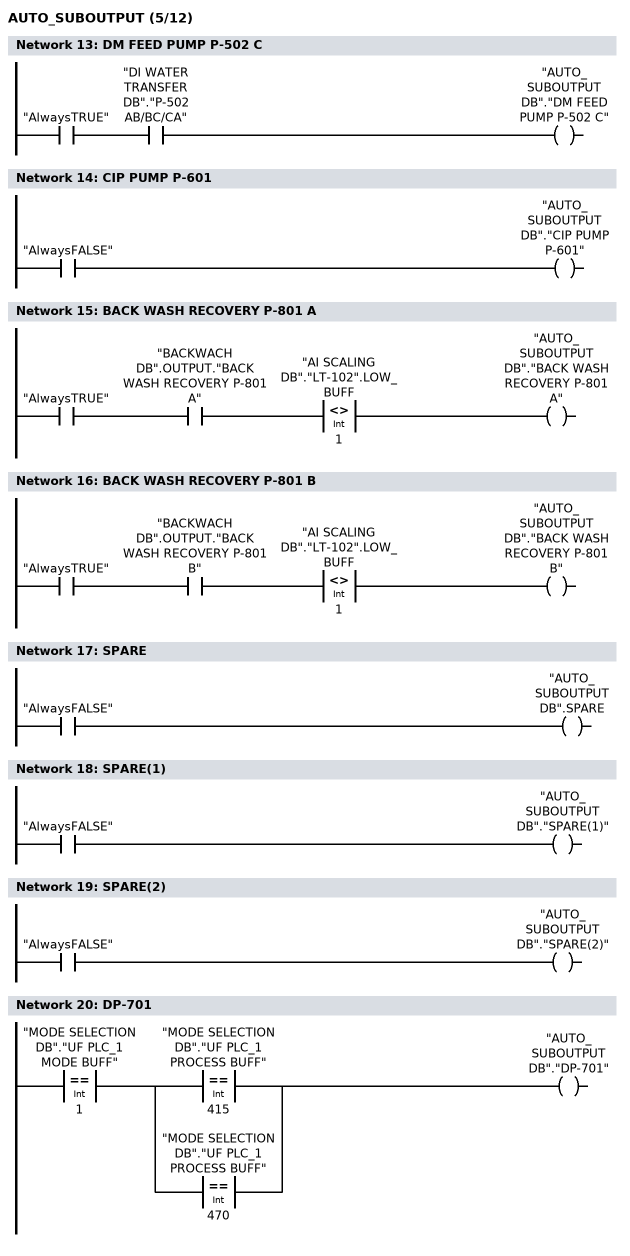
   RUNG wire#powerrail
      Contact( "AlwaysTRUE" )
      Contact( "DI WATER TRANSFER DB"."P-502 AB/BC/CA" )
      Coil( "AUTO_SUBOUTPUT DB"."DM FEED PUMP P-502 C" )
   END_RUNG
   // the same network as SCL:
   "AUTO_SUBOUTPUT DB"."DM FEED PUMP P-502 C" := "AlwaysTRUE" AND "DI WATER TRANSFER DB"."P-502 AB/BC/CA";
END_REGION

REGION Network 14: CIP PUMP P-601
   RUNG wire#powerrail
      Contact( "AlwaysFALSE" )
      Coil( "AUTO_SUBOUTPUT DB"."CIP PUMP P-601" )
   END_RUNG
   // the same network as SCL:
   "AUTO_SUBOUTPUT DB"."CIP PUMP P-601" := "AlwaysFALSE";
END_REGION

REGION Network 15: BACK WASH RECOVERY P-801 A
   RUNG wire#powerrail
      Contact( "AlwaysTRUE" )
      Contact( "BACKWACH DB".OUTPUT."BACK WASH RECOVERY P-801 A" )
      { S7_Templates := "SrcType := Int" } NE_Contact(in1 := "AI SCALING DB"."LT-102".LOW_BUFF, in2 := 1)
      Coil( "AUTO_SUBOUTPUT DB"."BACK WASH RECOVERY P-801 A" )
   END_RUNG
   // the same network as SCL:
   "AUTO_SUBOUTPUT DB"."BACK WASH RECOVERY P-801 A" := "AlwaysTRUE" AND "BACKWACH DB".OUTPUT."BACK WASH RECOVERY P-801 A" AND ("AI SCALING DB"."LT-102".LOW_BUFF <> 1);
END_REGION

REGION Network 16: BACK WASH RECOVERY P-801 B
   RUNG wire#powerrail
      Contact( "AlwaysTRUE" )
      Contact( "BACKWACH DB".OUTPUT."BACK WASH RECOVERY P-801 B" )
      { S7_Templates := "SrcType := Int" } NE_Contact(in1 := "AI SCALING DB"."LT-102".LOW_BUFF, in2 := 1)
      Coil( "AUTO_SUBOUTPUT DB"."BACK WASH RECOVERY P-801 B" )
   END_RUNG
   // the same network as SCL:
   "AUTO_SUBOUTPUT DB"."BACK WASH RECOVERY P-801 B" := "AlwaysTRUE" AND "BACKWACH DB".OUTPUT."BACK WASH RECOVERY P-801 B" AND ("AI SCALING DB"."LT-102".LOW_BUFF <> 1);
END_REGION

REGION Network 17: SPARE
   RUNG wire#powerrail
      Contact( "AlwaysFALSE" )
      Coil( "AUTO_SUBOUTPUT DB".SPARE )
   END_RUNG
   // the same network as SCL:
   "AUTO_SUBOUTPUT DB".SPARE := "AlwaysFALSE";
END_REGION

REGION Network 18: SPARE(1)
   RUNG wire#powerrail
      Contact( "AlwaysFALSE" )
      Coil( "AUTO_SUBOUTPUT DB"."SPARE(1)" )
   END_RUNG
   // the same network as SCL:
   "AUTO_SUBOUTPUT DB"."SPARE(1)" := "AlwaysFALSE";
END_REGION

REGION Network 19: SPARE(2)
   RUNG wire#powerrail
      Contact( "AlwaysFALSE" )
      Coil( "AUTO_SUBOUTPUT DB"."SPARE(2)" )
   END_RUNG
   // the same network as SCL:
   "AUTO_SUBOUTPUT DB"."SPARE(2)" := "AlwaysFALSE";
END_REGION

REGION Network 20: DP-701
   RUNG wire#powerrail
      { S7_Templates := "SrcType := Int" } EQ_Contact(in1 := "MODE SELECTION DB"."UF PLC_1 MODE BUFF", in2 := 1)
      wire#w1
      { S7_Templates := "SrcType := Int" } EQ_Contact(in1 := "MODE SELECTION DB"."UF PLC_1 PROCESS BUFF", in2 := 415)
      wire#w2
      Coil( "AUTO_SUBOUTPUT DB"."DP-701" )
   END_RUNG
   RUNG wire#w1
      { S7_Templates := "SrcType := Int" } EQ_Contact(in1 := "MODE SELECTION DB"."UF PLC_1 PROCESS BUFF", in2 := 470)
   END_RUNG wire#w2
   // the same network as SCL:
   "AUTO_SUBOUTPUT DB"."DP-701" := ("MODE SELECTION DB"."UF PLC_1 MODE BUFF" = 1) AND (("MODE SELECTION DB"."UF PLC_1 PROCESS BUFF" = 415) OR ("MODE SELECTION DB"."UF PLC_1 PROCESS BUFF" = 470));
END_REGION

REGION Network 21: DP-702
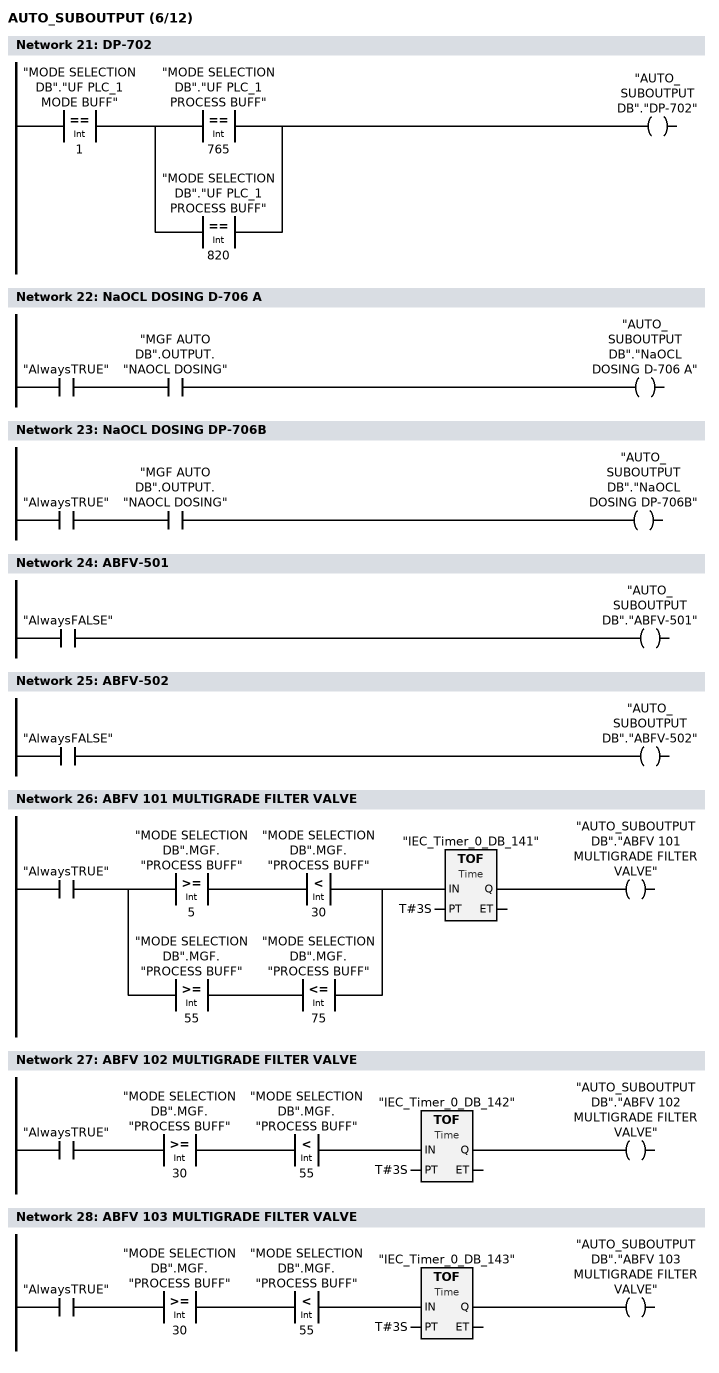
   RUNG wire#powerrail
      { S7_Templates := "SrcType := Int" } EQ_Contact(in1 := "MODE SELECTION DB"."UF PLC_1 MODE BUFF", in2 := 1)
      wire#w1
      { S7_Templates := "SrcType := Int" } EQ_Contact(in1 := "MODE SELECTION DB"."UF PLC_1 PROCESS BUFF", in2 := 765)
      wire#w2
      Coil( "AUTO_SUBOUTPUT DB"."DP-702" )
   END_RUNG
   RUNG wire#w1
      { S7_Templates := "SrcType := Int" } EQ_Contact(in1 := "MODE SELECTION DB"."UF PLC_1 PROCESS BUFF", in2 := 820)
   END_RUNG wire#w2
   // the same network as SCL:
   "AUTO_SUBOUTPUT DB"."DP-702" := ("MODE SELECTION DB"."UF PLC_1 MODE BUFF" = 1) AND (("MODE SELECTION DB"."UF PLC_1 PROCESS BUFF" = 765) OR ("MODE SELECTION DB"."UF PLC_1 PROCESS BUFF" = 820));
END_REGION

REGION Network 22: NaOCL DOSING D-706 A
   RUNG wire#powerrail
      Contact( "AlwaysTRUE" )
      Contact( "MGF AUTO DB".OUTPUT."NAOCL DOSING" )
      Coil( "AUTO_SUBOUTPUT DB"."NaOCL DOSING D-706 A" )
   END_RUNG
   // the same network as SCL:
   "AUTO_SUBOUTPUT DB"."NaOCL DOSING D-706 A" := "AlwaysTRUE" AND "MGF AUTO DB".OUTPUT."NAOCL DOSING";
END_REGION

REGION Network 23: NaOCL DOSING DP-706B
   RUNG wire#powerrail
      Contact( "AlwaysTRUE" )
      Contact( "MGF AUTO DB".OUTPUT."NAOCL DOSING" )
      Coil( "AUTO_SUBOUTPUT DB"."NaOCL DOSING DP-706B" )
   END_RUNG
   // the same network as SCL:
   "AUTO_SUBOUTPUT DB"."NaOCL DOSING DP-706B" := "AlwaysTRUE" AND "MGF AUTO DB".OUTPUT."NAOCL DOSING";
END_REGION

REGION Network 24: ABFV-501
   RUNG wire#powerrail
      Contact( "AlwaysFALSE" )
      Coil( "AUTO_SUBOUTPUT DB"."ABFV-501" )
   END_RUNG
   // the same network as SCL:
   "AUTO_SUBOUTPUT DB"."ABFV-501" := "AlwaysFALSE";
END_REGION

REGION Network 25: ABFV-502
   RUNG wire#powerrail
      Contact( "AlwaysFALSE" )
      Coil( "AUTO_SUBOUTPUT DB"."ABFV-502" )
   END_RUNG
   // the same network as SCL:
   "AUTO_SUBOUTPUT DB"."ABFV-502" := "AlwaysFALSE";
END_REGION

REGION Network 26: ABFV 101 MULTIGRADE FILTER VALVE
   RUNG wire#powerrail
      Contact( "AlwaysTRUE" )
      wire#w1
      { S7_Templates := "SrcType := Int" } GE_Contact(in1 := "MODE SELECTION DB".MGF."PROCESS BUFF", in2 := 5)
      { S7_Templates := "SrcType := Int" } LT_Contact(in1 := "MODE SELECTION DB".MGF."PROCESS BUFF", in2 := 30)
      wire#w2
      { S7_Templates := "time_type := Time" } "IEC_Timer_0_DB_141".TOF(pt := T#3S, et =>)
      Coil( "AUTO_SUBOUTPUT DB"."ABFV 101 MULTIGRADE FILTER VALVE" )
   END_RUNG
   RUNG wire#w1
      { S7_Templates := "SrcType := Int" } GE_Contact(in1 := "MODE SELECTION DB".MGF."PROCESS BUFF", in2 := 55)
      { S7_Templates := "SrcType := Int" } LE_Contact(in1 := "MODE SELECTION DB".MGF."PROCESS BUFF", in2 := 75)
   END_RUNG wire#w2
   // the same network as SCL:
   "IEC_Timer_0_DB_141".TOF(IN := "AlwaysTRUE" AND ((("MODE SELECTION DB".MGF."PROCESS BUFF" >= 5) AND ("MODE SELECTION DB".MGF."PROCESS BUFF" < 30)) OR (("MODE SELECTION DB".MGF."PROCESS BUFF" >= 55) AND ("MODE SELECTION DB".MGF."PROCESS BUFF" <= 75))),
                           PT := T#3S);
   "AUTO_SUBOUTPUT DB"."ABFV 101 MULTIGRADE FILTER VALVE" := "IEC_Timer_0_DB_141".Q;
END_REGION

REGION Network 27: ABFV 102 MULTIGRADE FILTER VALVE
   RUNG wire#powerrail
      Contact( "AlwaysTRUE" )
      { S7_Templates := "SrcType := Int" } GE_Contact(in1 := "MODE SELECTION DB".MGF."PROCESS BUFF", in2 := 30)
      { S7_Templates := "SrcType := Int" } LT_Contact(in1 := "MODE SELECTION DB".MGF."PROCESS BUFF", in2 := 55)
      { S7_Templates := "time_type := Time" } "IEC_Timer_0_DB_142".TOF(pt := T#3S, et =>)
      Coil( "AUTO_SUBOUTPUT DB"."ABFV 102 MULTIGRADE FILTER VALVE" )
   END_RUNG
   // the same network as SCL:
   "IEC_Timer_0_DB_142".TOF(IN := "AlwaysTRUE" AND ("MODE SELECTION DB".MGF."PROCESS BUFF" >= 30) AND ("MODE SELECTION DB".MGF."PROCESS BUFF" < 55),
                           PT := T#3S);
   "AUTO_SUBOUTPUT DB"."ABFV 102 MULTIGRADE FILTER VALVE" := "IEC_Timer_0_DB_142".Q;
END_REGION

REGION Network 28: ABFV 103 MULTIGRADE FILTER VALVE
   RUNG wire#powerrail
      Contact( "AlwaysTRUE" )
      { S7_Templates := "SrcType := Int" } GE_Contact(in1 := "MODE SELECTION DB".MGF."PROCESS BUFF", in2 := 30)
      { S7_Templates := "SrcType := Int" } LT_Contact(in1 := "MODE SELECTION DB".MGF."PROCESS BUFF", in2 := 55)
      { S7_Templates := "time_type := Time" } "IEC_Timer_0_DB_143".TOF(pt := T#3S, et =>)
      Coil( "AUTO_SUBOUTPUT DB"."ABFV 103 MULTIGRADE FILTER VALVE" )
   END_RUNG
   // the same network as SCL:
   "IEC_Timer_0_DB_143".TOF(IN := "AlwaysTRUE" AND ("MODE SELECTION DB".MGF."PROCESS BUFF" >= 30) AND ("MODE SELECTION DB".MGF."PROCESS BUFF" < 55),
                           PT := T#3S);
   "AUTO_SUBOUTPUT DB"."ABFV 103 MULTIGRADE FILTER VALVE" := "IEC_Timer_0_DB_143".Q;
END_REGION

REGION Network 29: ABFV 104 MULTIGRADE FILTER VALVE
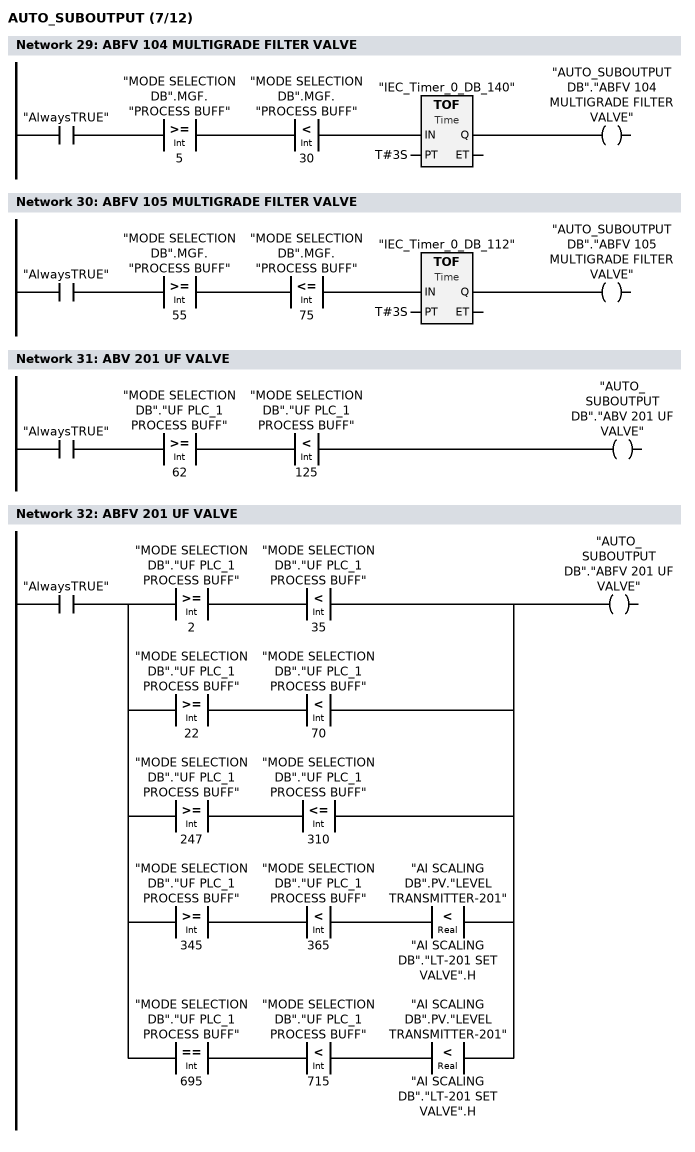
   RUNG wire#powerrail
      Contact( "AlwaysTRUE" )
      { S7_Templates := "SrcType := Int" } GE_Contact(in1 := "MODE SELECTION DB".MGF."PROCESS BUFF", in2 := 5)
      { S7_Templates := "SrcType := Int" } LT_Contact(in1 := "MODE SELECTION DB".MGF."PROCESS BUFF", in2 := 30)
      { S7_Templates := "time_type := Time" } "IEC_Timer_0_DB_140".TOF(pt := T#3S, et =>)
      Coil( "AUTO_SUBOUTPUT DB"."ABFV 104 MULTIGRADE FILTER VALVE" )
   END_RUNG
   // the same network as SCL:
   "IEC_Timer_0_DB_140".TOF(IN := "AlwaysTRUE" AND ("MODE SELECTION DB".MGF."PROCESS BUFF" >= 5) AND ("MODE SELECTION DB".MGF."PROCESS BUFF" < 30),
                           PT := T#3S);
   "AUTO_SUBOUTPUT DB"."ABFV 104 MULTIGRADE FILTER VALVE" := "IEC_Timer_0_DB_140".Q;
END_REGION

REGION Network 30: ABFV 105 MULTIGRADE FILTER VALVE
   RUNG wire#powerrail
      Contact( "AlwaysTRUE" )
      { S7_Templates := "SrcType := Int" } GE_Contact(in1 := "MODE SELECTION DB".MGF."PROCESS BUFF", in2 := 55)
      { S7_Templates := "SrcType := Int" } LE_Contact(in1 := "MODE SELECTION DB".MGF."PROCESS BUFF", in2 := 75)
      { S7_Templates := "time_type := Time" } "IEC_Timer_0_DB_112".TOF(pt := T#3S, et =>)
      Coil( "AUTO_SUBOUTPUT DB"."ABFV 105 MULTIGRADE FILTER VALVE" )
   END_RUNG
   // the same network as SCL:
   "IEC_Timer_0_DB_112".TOF(IN := "AlwaysTRUE" AND ("MODE SELECTION DB".MGF."PROCESS BUFF" >= 55) AND ("MODE SELECTION DB".MGF."PROCESS BUFF" <= 75),
                           PT := T#3S);
   "AUTO_SUBOUTPUT DB"."ABFV 105 MULTIGRADE FILTER VALVE" := "IEC_Timer_0_DB_112".Q;
END_REGION

REGION Network 31: ABV 201 UF VALVE
   RUNG wire#powerrail
      Contact( "AlwaysTRUE" )
      { S7_Templates := "SrcType := Int" } GE_Contact(in1 := "MODE SELECTION DB"."UF PLC_1 PROCESS BUFF", in2 := 62)
      { S7_Templates := "SrcType := Int" } LT_Contact(in1 := "MODE SELECTION DB"."UF PLC_1 PROCESS BUFF", in2 := 125)
      Coil( "AUTO_SUBOUTPUT DB"."ABV 201 UF VALVE" )
   END_RUNG
   // the same network as SCL:
   "AUTO_SUBOUTPUT DB"."ABV 201 UF VALVE" := "AlwaysTRUE" AND ("MODE SELECTION DB"."UF PLC_1 PROCESS BUFF" >= 62) AND ("MODE SELECTION DB"."UF PLC_1 PROCESS BUFF" < 125);
END_REGION

REGION Network 32: ABFV 201 UF VALVE
   RUNG wire#powerrail
      Contact( "AlwaysTRUE" )
      wire#w1
      { S7_Templates := "SrcType := Int" } GE_Contact(in1 := "MODE SELECTION DB"."UF PLC_1 PROCESS BUFF", in2 := 2)
      { S7_Templates := "SrcType := Int" } LT_Contact(in1 := "MODE SELECTION DB"."UF PLC_1 PROCESS BUFF", in2 := 35)
      wire#w2
      Coil( "AUTO_SUBOUTPUT DB"."ABFV 201 UF VALVE" )
   END_RUNG
   RUNG wire#w1
      { S7_Templates := "SrcType := Int" } GE_Contact(in1 := "MODE SELECTION DB"."UF PLC_1 PROCESS BUFF", in2 := 22)
      { S7_Templates := "SrcType := Int" } LT_Contact(in1 := "MODE SELECTION DB"."UF PLC_1 PROCESS BUFF", in2 := 70)
   END_RUNG wire#w2
   RUNG wire#w1
      { S7_Templates := "SrcType := Int" } GE_Contact(in1 := "MODE SELECTION DB"."UF PLC_1 PROCESS BUFF", in2 := 247)
      { S7_Templates := "SrcType := Int" } LE_Contact(in1 := "MODE SELECTION DB"."UF PLC_1 PROCESS BUFF", in2 := 310)
   END_RUNG wire#w2
   RUNG wire#w1
      { S7_Templates := "SrcType := Int" } GE_Contact(in1 := "MODE SELECTION DB"."UF PLC_1 PROCESS BUFF", in2 := 345)
      { S7_Templates := "SrcType := Int" } LT_Contact(in1 := "MODE SELECTION DB"."UF PLC_1 PROCESS BUFF", in2 := 365)
      { S7_Templates := "SrcType := Real" } LT_Contact(in1 := "AI SCALING DB".PV."LEVEL TRANSMITTER-201", in2 := "AI SCALING DB"."LT-201 SET VALVE".H)
   END_RUNG wire#w2
   RUNG wire#w1
      { S7_Templates := "SrcType := Int" } EQ_Contact(in1 := "MODE SELECTION DB"."UF PLC_1 PROCESS BUFF", in2 := 695)
      { S7_Templates := "SrcType := Int" } LT_Contact(in1 := "MODE SELECTION DB"."UF PLC_1 PROCESS BUFF", in2 := 715)
      { S7_Templates := "SrcType := Real" } LT_Contact(in1 := "AI SCALING DB".PV."LEVEL TRANSMITTER-201", in2 := "AI SCALING DB"."LT-201 SET VALVE".H)
   END_RUNG wire#w2
   // the same network as SCL:
   "AUTO_SUBOUTPUT DB"."ABFV 201 UF VALVE" := "AlwaysTRUE" AND ((("MODE SELECTION DB"."UF PLC_1 PROCESS BUFF" >= 2) AND ("MODE SELECTION DB"."UF PLC_1 PROCESS BUFF" < 35)) OR (("MODE SELECTION DB"."UF PLC_1 PROCESS BUFF" >= 22) AND ("MODE SELECTION DB"."UF PLC_1 PROCESS BUFF" < 70)) OR (("MODE SELECTION DB"."UF PLC_1 PROCESS BUFF" >= 247) AND ("MODE SELECTION DB"."UF PLC_1 PROCESS BUFF" <= 310)) OR (("MODE SELECTION DB"."UF PLC_1 PROCESS BUFF" >= 345) AND ("MODE SELECTION DB"."UF PLC_1 PROCESS BUFF" < 365) AND ("AI SCALING DB".PV."LEVEL TRANSMITTER-201" < "AI SCALING DB"."LT-201 SET VALVE".H)) OR (("MODE SELECTION DB"."UF PLC_1 PROCESS BUFF" = 695) AND ("MODE SELECTION DB"."UF PLC_1 PROCESS BUFF" < 715) AND ("AI SCALING DB".PV."LEVEL TRANSMITTER-201" < "AI SCALING DB"."LT-201 SET VALVE".H)));
END_REGION

REGION Network 33: ABFV 202 UF VALVE
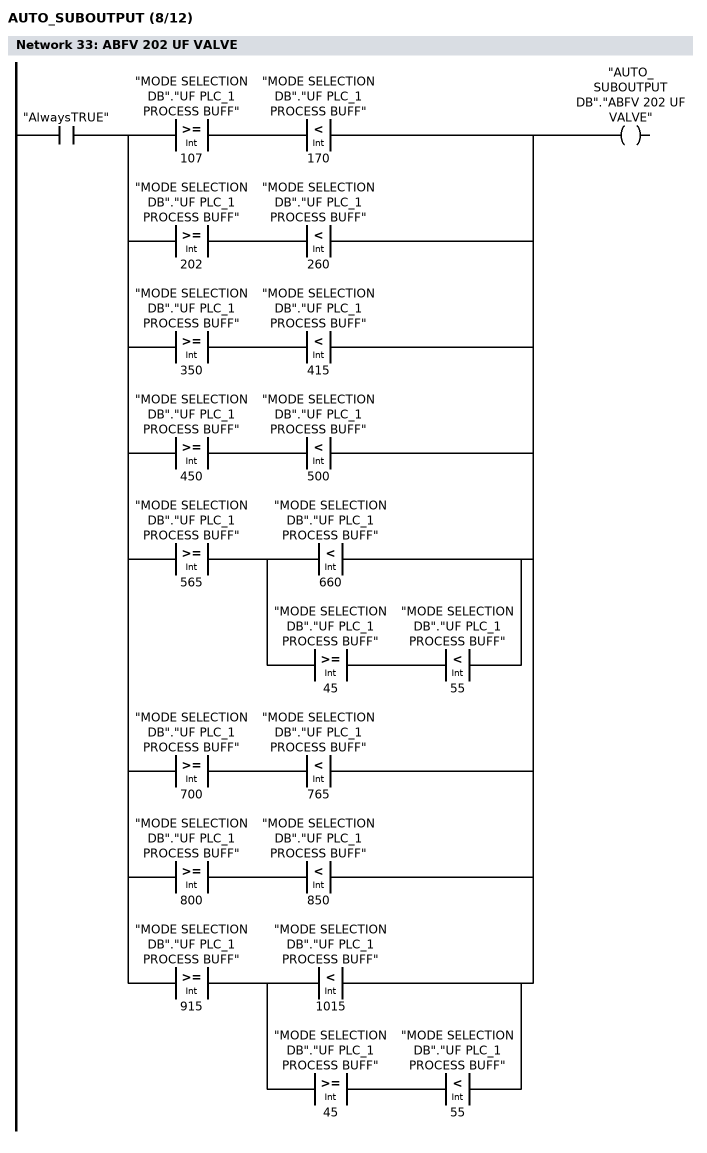
   RUNG wire#powerrail
      Contact( "AlwaysTRUE" )
      wire#w1
      { S7_Templates := "SrcType := Int" } GE_Contact(in1 := "MODE SELECTION DB"."UF PLC_1 PROCESS BUFF", in2 := 107)
      { S7_Templates := "SrcType := Int" } LT_Contact(in1 := "MODE SELECTION DB"."UF PLC_1 PROCESS BUFF", in2 := 170)
      wire#w2
      Coil( "AUTO_SUBOUTPUT DB"."ABFV 202 UF VALVE" )
   END_RUNG
   RUNG wire#w1
      { S7_Templates := "SrcType := Int" } GE_Contact(in1 := "MODE SELECTION DB"."UF PLC_1 PROCESS BUFF", in2 := 202)
      { S7_Templates := "SrcType := Int" } LT_Contact(in1 := "MODE SELECTION DB"."UF PLC_1 PROCESS BUFF", in2 := 260)
   END_RUNG wire#w2
   RUNG wire#w1
      { S7_Templates := "SrcType := Int" } GE_Contact(in1 := "MODE SELECTION DB"."UF PLC_1 PROCESS BUFF", in2 := 350)
      { S7_Templates := "SrcType := Int" } LT_Contact(in1 := "MODE SELECTION DB"."UF PLC_1 PROCESS BUFF", in2 := 415)
   END_RUNG wire#w2
   RUNG wire#w1
      { S7_Templates := "SrcType := Int" } GE_Contact(in1 := "MODE SELECTION DB"."UF PLC_1 PROCESS BUFF", in2 := 450)
      { S7_Templates := "SrcType := Int" } LT_Contact(in1 := "MODE SELECTION DB"."UF PLC_1 PROCESS BUFF", in2 := 500)
   END_RUNG wire#w2
   RUNG wire#w1
      { S7_Templates := "SrcType := Int" } GE_Contact(in1 := "MODE SELECTION DB"."UF PLC_1 PROCESS BUFF", in2 := 565)
      wire#w3
      { S7_Templates := "SrcType := Int" } LT_Contact(in1 := "MODE SELECTION DB"."UF PLC_1 PROCESS BUFF", in2 := 660)
   END_RUNG wire#w2
   RUNG wire#w3
      { S7_Templates := "SrcType := Int" } GE_Contact(in1 := "MODE SELECTION DB"."UF PLC_1 PROCESS BUFF", in2 := 45)
      { S7_Templates := "SrcType := Int" } LT_Contact(in1 := "MODE SELECTION DB"."UF PLC_1 PROCESS BUFF", in2 := 55)
   END_RUNG wire#w2
   RUNG wire#w1
      { S7_Templates := "SrcType := Int" } GE_Contact(in1 := "MODE SELECTION DB"."UF PLC_1 PROCESS BUFF", in2 := 700)
      { S7_Templates := "SrcType := Int" } LT_Contact(in1 := "MODE SELECTION DB"."UF PLC_1 PROCESS BUFF", in2 := 765)
   END_RUNG wire#w2
   RUNG wire#w1
      { S7_Templates := "SrcType := Int" } GE_Contact(in1 := "MODE SELECTION DB"."UF PLC_1 PROCESS BUFF", in2 := 800)
      { S7_Templates := "SrcType := Int" } LT_Contact(in1 := "MODE SELECTION DB"."UF PLC_1 PROCESS BUFF", in2 := 850)
   END_RUNG wire#w2
   RUNG wire#w1
      { S7_Templates := "SrcType := Int" } GE_Contact(in1 := "MODE SELECTION DB"."UF PLC_1 PROCESS BUFF", in2 := 915)
      wire#w4
      { S7_Templates := "SrcType := Int" } LT_Contact(in1 := "MODE SELECTION DB"."UF PLC_1 PROCESS BUFF", in2 := 1015)
   END_RUNG wire#w2
   RUNG wire#w4
      { S7_Templates := "SrcType := Int" } GE_Contact(in1 := "MODE SELECTION DB"."UF PLC_1 PROCESS BUFF", in2 := 45)
      { S7_Templates := "SrcType := Int" } LT_Contact(in1 := "MODE SELECTION DB"."UF PLC_1 PROCESS BUFF", in2 := 55)
   END_RUNG wire#w2
   // the same network as SCL:
   "AUTO_SUBOUTPUT DB"."ABFV 202 UF VALVE" := "AlwaysTRUE" AND ((("MODE SELECTION DB"."UF PLC_1 PROCESS BUFF" >= 107) AND ("MODE SELECTION DB"."UF PLC_1 PROCESS BUFF" < 170)) OR (("MODE SELECTION DB"."UF PLC_1 PROCESS BUFF" >= 202) AND ("MODE SELECTION DB"."UF PLC_1 PROCESS BUFF" < 260)) OR (("MODE SELECTION DB"."UF PLC_1 PROCESS BUFF" >= 350) AND ("MODE SELECTION DB"."UF PLC_1 PROCESS BUFF" < 415)) OR (("MODE SELECTION DB"."UF PLC_1 PROCESS BUFF" >= 450) AND ("MODE SELECTION DB"."UF PLC_1 PROCESS BUFF" < 500)) OR (("MODE SELECTION DB"."UF PLC_1 PROCESS BUFF" >= 565) AND (("MODE SELECTION DB"."UF PLC_1 PROCESS BUFF" < 660) OR (("MODE SELECTION DB"."UF PLC_1 PROCESS BUFF" >= 45) AND ("MODE SELECTION DB"."UF PLC_1 PROCESS BUFF" < 55)))) OR (("MODE SELECTION DB"."UF PLC_1 PROCESS BUFF" >= 700) AND ("MODE SELECTION DB"."UF PLC_1 PROCESS BUFF" < 765)) OR (("MODE SELECTION DB"."UF PLC_1 PROCESS BUFF" >= 800) AND ("MODE SELECTION DB"."UF PLC_1 PROCESS BUFF" < 850)) OR (("MODE SELECTION DB"."UF PLC_1 PROCESS BUFF" >= 915) AND (("MODE SELECTION DB"."UF PLC_1 PROCESS BUFF" < 1015) OR (("MODE SELECTION DB"."UF PLC_1 PROCESS BUFF" >= 45) AND ("MODE SELECTION DB"."UF PLC_1 PROCESS BUFF" < 55)))));
END_REGION

REGION Network 34: ABFV 203 UF VALVE
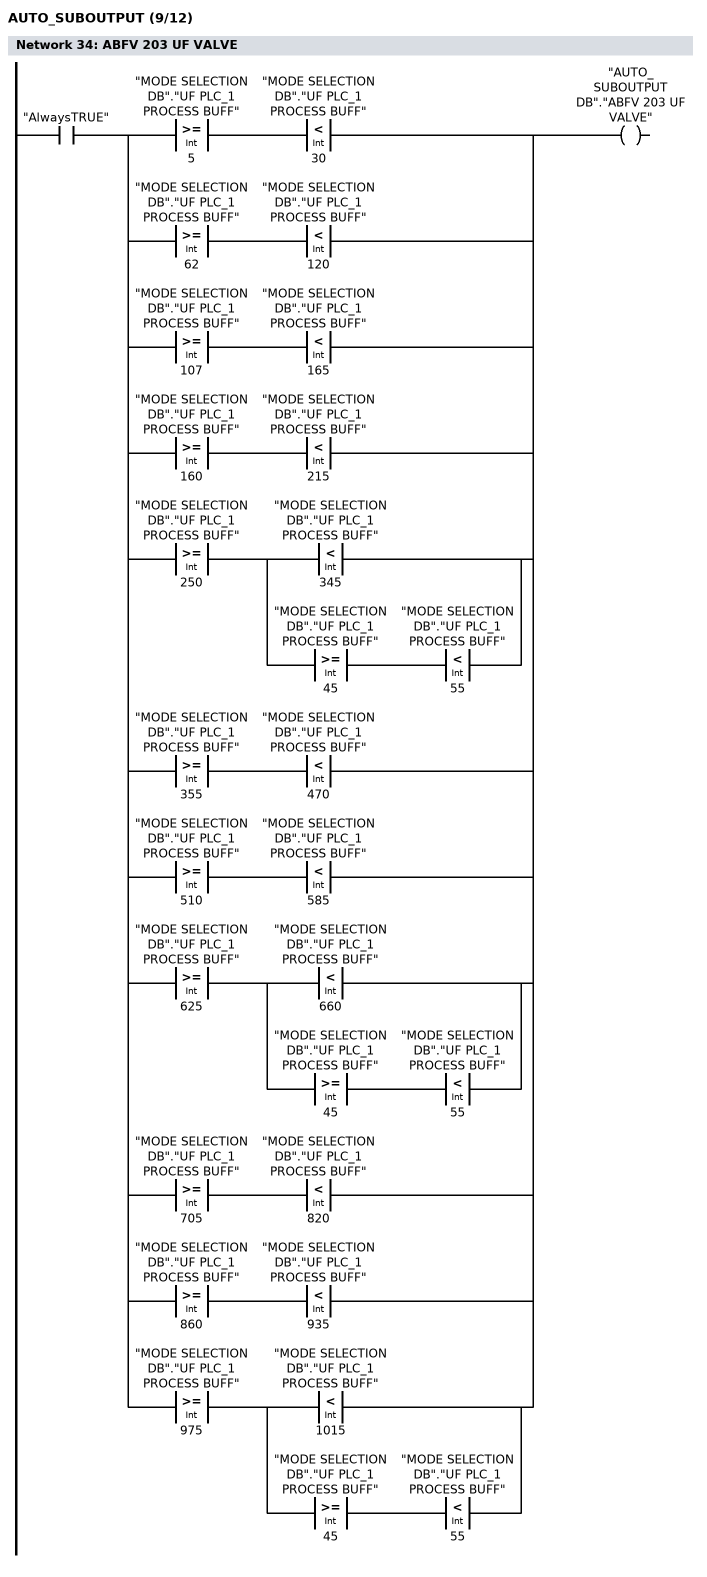
   RUNG wire#powerrail
      Contact( "AlwaysTRUE" )
      wire#w1
      { S7_Templates := "SrcType := Int" } GE_Contact(in1 := "MODE SELECTION DB"."UF PLC_1 PROCESS BUFF", in2 := 5)
      { S7_Templates := "SrcType := Int" } LT_Contact(in1 := "MODE SELECTION DB"."UF PLC_1 PROCESS BUFF", in2 := 30)
      wire#w2
      Coil( "AUTO_SUBOUTPUT DB"."ABFV 203 UF VALVE" )
   END_RUNG
   RUNG wire#w1
      { S7_Templates := "SrcType := Int" } GE_Contact(in1 := "MODE SELECTION DB"."UF PLC_1 PROCESS BUFF", in2 := 62)
      { S7_Templates := "SrcType := Int" } LT_Contact(in1 := "MODE SELECTION DB"."UF PLC_1 PROCESS BUFF", in2 := 120)
   END_RUNG wire#w2
   RUNG wire#w1
      { S7_Templates := "SrcType := Int" } GE_Contact(in1 := "MODE SELECTION DB"."UF PLC_1 PROCESS BUFF", in2 := 107)
      { S7_Templates := "SrcType := Int" } LT_Contact(in1 := "MODE SELECTION DB"."UF PLC_1 PROCESS BUFF", in2 := 165)
   END_RUNG wire#w2
   RUNG wire#w1
      { S7_Templates := "SrcType := Int" } GE_Contact(in1 := "MODE SELECTION DB"."UF PLC_1 PROCESS BUFF", in2 := 160)
      { S7_Templates := "SrcType := Int" } LT_Contact(in1 := "MODE SELECTION DB"."UF PLC_1 PROCESS BUFF", in2 := 215)
   END_RUNG wire#w2
   RUNG wire#w1
      { S7_Templates := "SrcType := Int" } GE_Contact(in1 := "MODE SELECTION DB"."UF PLC_1 PROCESS BUFF", in2 := 250)
      wire#w3
      { S7_Templates := "SrcType := Int" } LT_Contact(in1 := "MODE SELECTION DB"."UF PLC_1 PROCESS BUFF", in2 := 345)
   END_RUNG wire#w2
   RUNG wire#w3
      { S7_Templates := "SrcType := Int" } GE_Contact(in1 := "MODE SELECTION DB"."UF PLC_1 PROCESS BUFF", in2 := 45)
      { S7_Templates := "SrcType := Int" } LT_Contact(in1 := "MODE SELECTION DB"."UF PLC_1 PROCESS BUFF", in2 := 55)
   END_RUNG wire#w2
   RUNG wire#w1
      { S7_Templates := "SrcType := Int" } GE_Contact(in1 := "MODE SELECTION DB"."UF PLC_1 PROCESS BUFF", in2 := 355)
      { S7_Templates := "SrcType := Int" } LT_Contact(in1 := "MODE SELECTION DB"."UF PLC_1 PROCESS BUFF", in2 := 470)
   END_RUNG wire#w2
   RUNG wire#w1
      { S7_Templates := "SrcType := Int" } GE_Contact(in1 := "MODE SELECTION DB"."UF PLC_1 PROCESS BUFF", in2 := 510)
      { S7_Templates := "SrcType := Int" } LT_Contact(in1 := "MODE SELECTION DB"."UF PLC_1 PROCESS BUFF", in2 := 585)
   END_RUNG wire#w2
   RUNG wire#w1
      { S7_Templates := "SrcType := Int" } GE_Contact(in1 := "MODE SELECTION DB"."UF PLC_1 PROCESS BUFF", in2 := 625)
      wire#w4
      { S7_Templates := "SrcType := Int" } LT_Contact(in1 := "MODE SELECTION DB"."UF PLC_1 PROCESS BUFF", in2 := 660)
   END_RUNG wire#w2
   RUNG wire#w4
      { S7_Templates := "SrcType := Int" } GE_Contact(in1 := "MODE SELECTION DB"."UF PLC_1 PROCESS BUFF", in2 := 45)
      { S7_Templates := "SrcType := Int" } LT_Contact(in1 := "MODE SELECTION DB"."UF PLC_1 PROCESS BUFF", in2 := 55)
   END_RUNG wire#w2
   RUNG wire#w1
      { S7_Templates := "SrcType := Int" } GE_Contact(in1 := "MODE SELECTION DB"."UF PLC_1 PROCESS BUFF", in2 := 705)
      { S7_Templates := "SrcType := Int" } LT_Contact(in1 := "MODE SELECTION DB"."UF PLC_1 PROCESS BUFF", in2 := 820)
   END_RUNG wire#w2
   RUNG wire#w1
      { S7_Templates := "SrcType := Int" } GE_Contact(in1 := "MODE SELECTION DB"."UF PLC_1 PROCESS BUFF", in2 := 860)
      { S7_Templates := "SrcType := Int" } LT_Contact(in1 := "MODE SELECTION DB"."UF PLC_1 PROCESS BUFF", in2 := 935)
   END_RUNG wire#w2
   RUNG wire#w1
      { S7_Templates := "SrcType := Int" } GE_Contact(in1 := "MODE SELECTION DB"."UF PLC_1 PROCESS BUFF", in2 := 975)
      wire#w5
      { S7_Templates := "SrcType := Int" } LT_Contact(in1 := "MODE SELECTION DB"."UF PLC_1 PROCESS BUFF", in2 := 1015)
   END_RUNG wire#w2
   RUNG wire#w5
      { S7_Templates := "SrcType := Int" } GE_Contact(in1 := "MODE SELECTION DB"."UF PLC_1 PROCESS BUFF", in2 := 45)
      { S7_Templates := "SrcType := Int" } LT_Contact(in1 := "MODE SELECTION DB"."UF PLC_1 PROCESS BUFF", in2 := 55)
   END_RUNG wire#w2
   // the same network as SCL:
   "AUTO_SUBOUTPUT DB"."ABFV 203 UF VALVE" := "AlwaysTRUE" AND ((("MODE SELECTION DB"."UF PLC_1 PROCESS BUFF" >= 5) AND ("MODE SELECTION DB"."UF PLC_1 PROCESS BUFF" < 30)) OR (("MODE SELECTION DB"."UF PLC_1 PROCESS BUFF" >= 62) AND ("MODE SELECTION DB"."UF PLC_1 PROCESS BUFF" < 120)) OR (("MODE SELECTION DB"."UF PLC_1 PROCESS BUFF" >= 107) AND ("MODE SELECTION DB"."UF PLC_1 PROCESS BUFF" < 165)) OR (("MODE SELECTION DB"."UF PLC_1 PROCESS BUFF" >= 160) AND ("MODE SELECTION DB"."UF PLC_1 PROCESS BUFF" < 215)) OR (("MODE SELECTION DB"."UF PLC_1 PROCESS BUFF" >= 250) AND (("MODE SELECTION DB"."UF PLC_1 PROCESS BUFF" < 345) OR (("MODE SELECTION DB"."UF PLC_1 PROCESS BUFF" >= 45) AND ("MODE SELECTION DB"."UF PLC_1 PROCESS BUFF" < 55)))) OR (("MODE SELECTION DB"."UF PLC_1 PROCESS BUFF" >= 355) AND ("MODE SELECTION DB"."UF PLC_1 PROCESS BUFF" < 470)) OR (("MODE SELECTION DB"."UF PLC_1 PROCESS BUFF" >= 510) AND ("MODE SELECTION DB"."UF PLC_1 PROCESS BUFF" < 585)) OR (("MODE SELECTION DB"."UF PLC_1 PROCESS BUFF" >= 625) AND (("MODE SELECTION DB"."UF PLC_1 PROCESS BUFF" < 660) OR (("MODE SELECTION DB"."UF PLC_1 PROCESS BUFF" >= 45) AND ("MODE SELECTION DB"."UF PLC_1 PROCESS BUFF" < 55)))) OR (("MODE SELECTION DB"."UF PLC_1 PROCESS BUFF" >= 705) AND ("MODE SELECTION DB"."UF PLC_1 PROCESS BUFF" < 820)) OR (("MODE SELECTION DB"."UF PLC_1 PROCESS BUFF" >= 860) AND ("MODE SELECTION DB"."UF PLC_1 PROCESS BUFF" < 935)) OR (("MODE SELECTION DB"."UF PLC_1 PROCESS BUFF" >= 975) AND (("MODE SELECTION DB"."UF PLC_1 PROCESS BUFF" < 1015) OR (("MODE SELECTION DB"."UF PLC_1 PROCESS BUFF" >= 45) AND ("MODE SELECTION DB"."UF PLC_1 PROCESS BUFF" < 55)))));
END_REGION

REGION Network 35: ABFV 204 UF VALVE
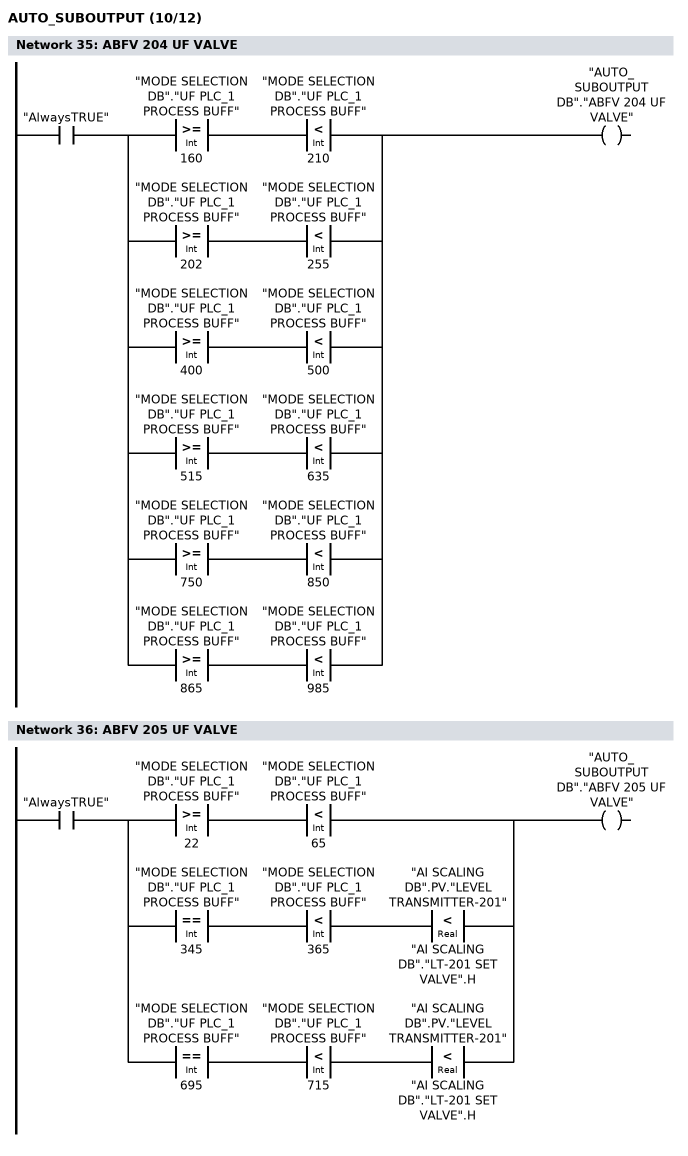
   RUNG wire#powerrail
      Contact( "AlwaysTRUE" )
      wire#w1
      { S7_Templates := "SrcType := Int" } GE_Contact(in1 := "MODE SELECTION DB"."UF PLC_1 PROCESS BUFF", in2 := 160)
      { S7_Templates := "SrcType := Int" } LT_Contact(in1 := "MODE SELECTION DB"."UF PLC_1 PROCESS BUFF", in2 := 210)
      wire#w2
      Coil( "AUTO_SUBOUTPUT DB"."ABFV 204 UF VALVE" )
   END_RUNG
   RUNG wire#w1
      { S7_Templates := "SrcType := Int" } GE_Contact(in1 := "MODE SELECTION DB"."UF PLC_1 PROCESS BUFF", in2 := 202)
      { S7_Templates := "SrcType := Int" } LT_Contact(in1 := "MODE SELECTION DB"."UF PLC_1 PROCESS BUFF", in2 := 255)
   END_RUNG wire#w2
   RUNG wire#w1
      { S7_Templates := "SrcType := Int" } GE_Contact(in1 := "MODE SELECTION DB"."UF PLC_1 PROCESS BUFF", in2 := 400)
      { S7_Templates := "SrcType := Int" } LT_Contact(in1 := "MODE SELECTION DB"."UF PLC_1 PROCESS BUFF", in2 := 500)
   END_RUNG wire#w2
   RUNG wire#w1
      { S7_Templates := "SrcType := Int" } GE_Contact(in1 := "MODE SELECTION DB"."UF PLC_1 PROCESS BUFF", in2 := 515)
      { S7_Templates := "SrcType := Int" } LT_Contact(in1 := "MODE SELECTION DB"."UF PLC_1 PROCESS BUFF", in2 := 635)
   END_RUNG wire#w2
   RUNG wire#w1
      { S7_Templates := "SrcType := Int" } GE_Contact(in1 := "MODE SELECTION DB"."UF PLC_1 PROCESS BUFF", in2 := 750)
      { S7_Templates := "SrcType := Int" } LT_Contact(in1 := "MODE SELECTION DB"."UF PLC_1 PROCESS BUFF", in2 := 850)
   END_RUNG wire#w2
   RUNG wire#w1
      { S7_Templates := "SrcType := Int" } GE_Contact(in1 := "MODE SELECTION DB"."UF PLC_1 PROCESS BUFF", in2 := 865)
      { S7_Templates := "SrcType := Int" } LT_Contact(in1 := "MODE SELECTION DB"."UF PLC_1 PROCESS BUFF", in2 := 985)
   END_RUNG wire#w2
   // the same network as SCL:
   "AUTO_SUBOUTPUT DB"."ABFV 204 UF VALVE" := "AlwaysTRUE" AND ((("MODE SELECTION DB"."UF PLC_1 PROCESS BUFF" >= 160) AND ("MODE SELECTION DB"."UF PLC_1 PROCESS BUFF" < 210)) OR (("MODE SELECTION DB"."UF PLC_1 PROCESS BUFF" >= 202) AND ("MODE SELECTION DB"."UF PLC_1 PROCESS BUFF" < 255)) OR (("MODE SELECTION DB"."UF PLC_1 PROCESS BUFF" >= 400) AND ("MODE SELECTION DB"."UF PLC_1 PROCESS BUFF" < 500)) OR (("MODE SELECTION DB"."UF PLC_1 PROCESS BUFF" >= 515) AND ("MODE SELECTION DB"."UF PLC_1 PROCESS BUFF" < 635)) OR (("MODE SELECTION DB"."UF PLC_1 PROCESS BUFF" >= 750) AND ("MODE SELECTION DB"."UF PLC_1 PROCESS BUFF" < 850)) OR (("MODE SELECTION DB"."UF PLC_1 PROCESS BUFF" >= 865) AND ("MODE SELECTION DB"."UF PLC_1 PROCESS BUFF" < 985)));
END_REGION

REGION Network 36: ABFV 205 UF VALVE
   RUNG wire#powerrail
      Contact( "AlwaysTRUE" )
      wire#w1
      { S7_Templates := "SrcType := Int" } GE_Contact(in1 := "MODE SELECTION DB"."UF PLC_1 PROCESS BUFF", in2 := 22)
      { S7_Templates := "SrcType := Int" } LT_Contact(in1 := "MODE SELECTION DB"."UF PLC_1 PROCESS BUFF", in2 := 65)
      wire#w2
      Coil( "AUTO_SUBOUTPUT DB"."ABFV 205 UF VALVE" )
   END_RUNG
   RUNG wire#w1
      { S7_Templates := "SrcType := Int" } EQ_Contact(in1 := "MODE SELECTION DB"."UF PLC_1 PROCESS BUFF", in2 := 345)
      { S7_Templates := "SrcType := Int" } LT_Contact(in1 := "MODE SELECTION DB"."UF PLC_1 PROCESS BUFF", in2 := 365)
      { S7_Templates := "SrcType := Real" } LT_Contact(in1 := "AI SCALING DB".PV."LEVEL TRANSMITTER-201", in2 := "AI SCALING DB"."LT-201 SET VALVE".H)
   END_RUNG wire#w2
   RUNG wire#w1
      { S7_Templates := "SrcType := Int" } EQ_Contact(in1 := "MODE SELECTION DB"."UF PLC_1 PROCESS BUFF", in2 := 695)
      { S7_Templates := "SrcType := Int" } LT_Contact(in1 := "MODE SELECTION DB"."UF PLC_1 PROCESS BUFF", in2 := 715)
      { S7_Templates := "SrcType := Real" } LT_Contact(in1 := "AI SCALING DB".PV."LEVEL TRANSMITTER-201", in2 := "AI SCALING DB"."LT-201 SET VALVE".H)
   END_RUNG wire#w2
   // the same network as SCL:
   "AUTO_SUBOUTPUT DB"."ABFV 205 UF VALVE" := "AlwaysTRUE" AND ((("MODE SELECTION DB"."UF PLC_1 PROCESS BUFF" >= 22) AND ("MODE SELECTION DB"."UF PLC_1 PROCESS BUFF" < 65)) OR (("MODE SELECTION DB"."UF PLC_1 PROCESS BUFF" = 345) AND ("MODE SELECTION DB"."UF PLC_1 PROCESS BUFF" < 365) AND ("AI SCALING DB".PV."LEVEL TRANSMITTER-201" < "AI SCALING DB"."LT-201 SET VALVE".H)) OR (("MODE SELECTION DB"."UF PLC_1 PROCESS BUFF" = 695) AND ("MODE SELECTION DB"."UF PLC_1 PROCESS BUFF" < 715) AND ("AI SCALING DB".PV."LEVEL TRANSMITTER-201" < "AI SCALING DB"."LT-201 SET VALVE".H)));
END_REGION

REGION Network 37: ABFV 206 UF VALVE
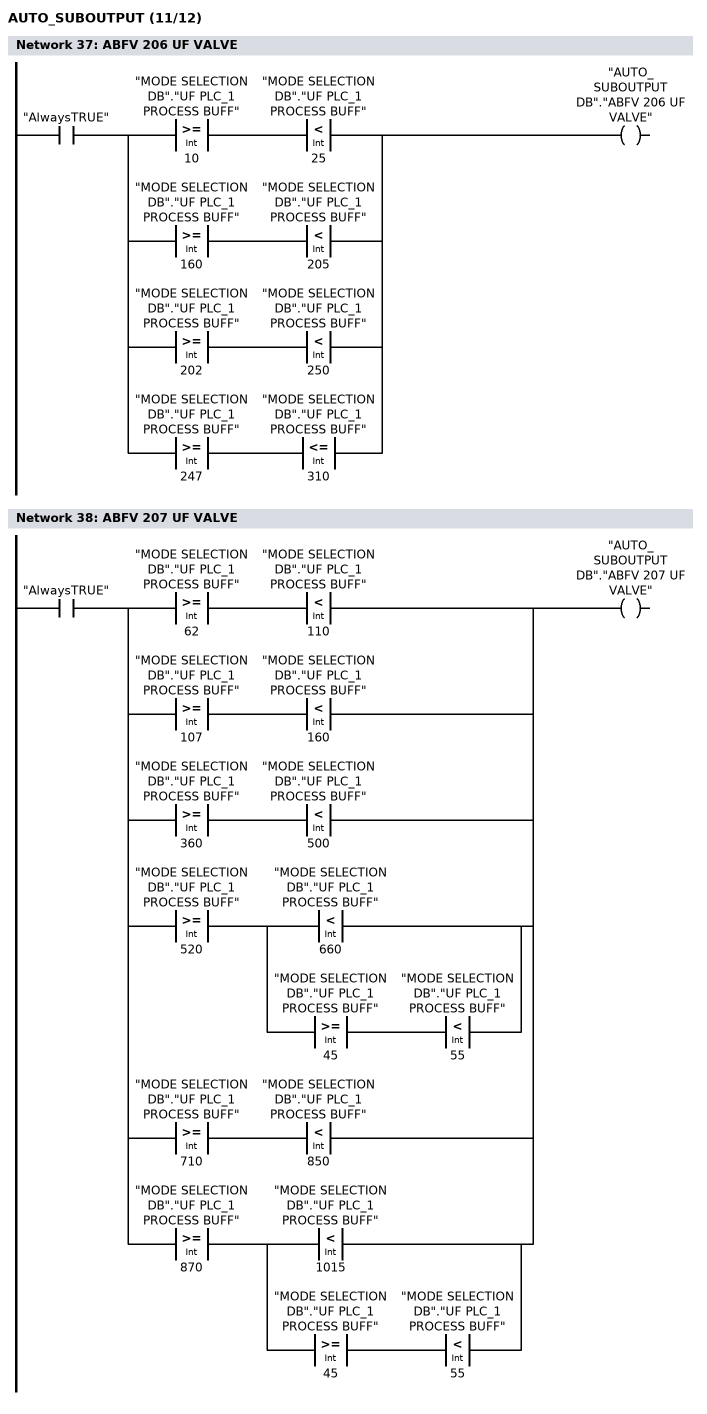
   RUNG wire#powerrail
      Contact( "AlwaysTRUE" )
      wire#w1
      { S7_Templates := "SrcType := Int" } GE_Contact(in1 := "MODE SELECTION DB"."UF PLC_1 PROCESS BUFF", in2 := 10)
      { S7_Templates := "SrcType := Int" } LT_Contact(in1 := "MODE SELECTION DB"."UF PLC_1 PROCESS BUFF", in2 := 25)
      wire#w2
      Coil( "AUTO_SUBOUTPUT DB"."ABFV 206 UF VALVE" )
   END_RUNG
   RUNG wire#w1
      { S7_Templates := "SrcType := Int" } GE_Contact(in1 := "MODE SELECTION DB"."UF PLC_1 PROCESS BUFF", in2 := 160)
      { S7_Templates := "SrcType := Int" } LT_Contact(in1 := "MODE SELECTION DB"."UF PLC_1 PROCESS BUFF", in2 := 205)
   END_RUNG wire#w2
   RUNG wire#w1
      { S7_Templates := "SrcType := Int" } GE_Contact(in1 := "MODE SELECTION DB"."UF PLC_1 PROCESS BUFF", in2 := 202)
      { S7_Templates := "SrcType := Int" } LT_Contact(in1 := "MODE SELECTION DB"."UF PLC_1 PROCESS BUFF", in2 := 250)
   END_RUNG wire#w2
   RUNG wire#w1
      { S7_Templates := "SrcType := Int" } GE_Contact(in1 := "MODE SELECTION DB"."UF PLC_1 PROCESS BUFF", in2 := 247)
      { S7_Templates := "SrcType := Int" } LE_Contact(in1 := "MODE SELECTION DB"."UF PLC_1 PROCESS BUFF", in2 := 310)
   END_RUNG wire#w2
   // the same network as SCL:
   "AUTO_SUBOUTPUT DB"."ABFV 206 UF VALVE" := "AlwaysTRUE" AND ((("MODE SELECTION DB"."UF PLC_1 PROCESS BUFF" >= 10) AND ("MODE SELECTION DB"."UF PLC_1 PROCESS BUFF" < 25)) OR (("MODE SELECTION DB"."UF PLC_1 PROCESS BUFF" >= 160) AND ("MODE SELECTION DB"."UF PLC_1 PROCESS BUFF" < 205)) OR (("MODE SELECTION DB"."UF PLC_1 PROCESS BUFF" >= 202) AND ("MODE SELECTION DB"."UF PLC_1 PROCESS BUFF" < 250)) OR (("MODE SELECTION DB"."UF PLC_1 PROCESS BUFF" >= 247) AND ("MODE SELECTION DB"."UF PLC_1 PROCESS BUFF" <= 310)));
END_REGION

REGION Network 38: ABFV 207 UF VALVE
   RUNG wire#powerrail
      Contact( "AlwaysTRUE" )
      wire#w1
      { S7_Templates := "SrcType := Int" } GE_Contact(in1 := "MODE SELECTION DB"."UF PLC_1 PROCESS BUFF", in2 := 62)
      { S7_Templates := "SrcType := Int" } LT_Contact(in1 := "MODE SELECTION DB"."UF PLC_1 PROCESS BUFF", in2 := 110)
      wire#w2
      Coil( "AUTO_SUBOUTPUT DB"."ABFV 207 UF VALVE" )
   END_RUNG
   RUNG wire#w1
      { S7_Templates := "SrcType := Int" } GE_Contact(in1 := "MODE SELECTION DB"."UF PLC_1 PROCESS BUFF", in2 := 107)
      { S7_Templates := "SrcType := Int" } LT_Contact(in1 := "MODE SELECTION DB"."UF PLC_1 PROCESS BUFF", in2 := 160)
   END_RUNG wire#w2
   RUNG wire#w1
      { S7_Templates := "SrcType := Int" } GE_Contact(in1 := "MODE SELECTION DB"."UF PLC_1 PROCESS BUFF", in2 := 360)
      { S7_Templates := "SrcType := Int" } LT_Contact(in1 := "MODE SELECTION DB"."UF PLC_1 PROCESS BUFF", in2 := 500)
   END_RUNG wire#w2
   RUNG wire#w1
      { S7_Templates := "SrcType := Int" } GE_Contact(in1 := "MODE SELECTION DB"."UF PLC_1 PROCESS BUFF", in2 := 520)
      wire#w3
      { S7_Templates := "SrcType := Int" } LT_Contact(in1 := "MODE SELECTION DB"."UF PLC_1 PROCESS BUFF", in2 := 660)
   END_RUNG wire#w2
   RUNG wire#w3
      { S7_Templates := "SrcType := Int" } GE_Contact(in1 := "MODE SELECTION DB"."UF PLC_1 PROCESS BUFF", in2 := 45)
      { S7_Templates := "SrcType := Int" } LT_Contact(in1 := "MODE SELECTION DB"."UF PLC_1 PROCESS BUFF", in2 := 55)
   END_RUNG wire#w2
   RUNG wire#w1
      { S7_Templates := "SrcType := Int" } GE_Contact(in1 := "MODE SELECTION DB"."UF PLC_1 PROCESS BUFF", in2 := 710)
      { S7_Templates := "SrcType := Int" } LT_Contact(in1 := "MODE SELECTION DB"."UF PLC_1 PROCESS BUFF", in2 := 850)
   END_RUNG wire#w2
   RUNG wire#w1
      { S7_Templates := "SrcType := Int" } GE_Contact(in1 := "MODE SELECTION DB"."UF PLC_1 PROCESS BUFF", in2 := 870)
      wire#w4
      { S7_Templates := "SrcType := Int" } LT_Contact(in1 := "MODE SELECTION DB"."UF PLC_1 PROCESS BUFF", in2 := 1015)
   END_RUNG wire#w2
   RUNG wire#w4
      { S7_Templates := "SrcType := Int" } GE_Contact(in1 := "MODE SELECTION DB"."UF PLC_1 PROCESS BUFF", in2 := 45)
      { S7_Templates := "SrcType := Int" } LT_Contact(in1 := "MODE SELECTION DB"."UF PLC_1 PROCESS BUFF", in2 := 55)
   END_RUNG wire#w2
   // the same network as SCL:
   "AUTO_SUBOUTPUT DB"."ABFV 207 UF VALVE" := "AlwaysTRUE" AND ((("MODE SELECTION DB"."UF PLC_1 PROCESS BUFF" >= 62) AND ("MODE SELECTION DB"."UF PLC_1 PROCESS BUFF" < 110)) OR (("MODE SELECTION DB"."UF PLC_1 PROCESS BUFF" >= 107) AND ("MODE SELECTION DB"."UF PLC_1 PROCESS BUFF" < 160)) OR (("MODE SELECTION DB"."UF PLC_1 PROCESS BUFF" >= 360) AND ("MODE SELECTION DB"."UF PLC_1 PROCESS BUFF" < 500)) OR (("MODE SELECTION DB"."UF PLC_1 PROCESS BUFF" >= 520) AND (("MODE SELECTION DB"."UF PLC_1 PROCESS BUFF" < 660) OR (("MODE SELECTION DB"."UF PLC_1 PROCESS BUFF" >= 45) AND ("MODE SELECTION DB"."UF PLC_1 PROCESS BUFF" < 55)))) OR (("MODE SELECTION DB"."UF PLC_1 PROCESS BUFF" >= 710) AND ("MODE SELECTION DB"."UF PLC_1 PROCESS BUFF" < 850)) OR (("MODE SELECTION DB"."UF PLC_1 PROCESS BUFF" >= 870) AND (("MODE SELECTION DB"."UF PLC_1 PROCESS BUFF" < 1015) OR (("MODE SELECTION DB"."UF PLC_1 PROCESS BUFF" >= 45) AND ("MODE SELECTION DB"."UF PLC_1 PROCESS BUFF" < 55)))));
END_REGION

REGION Network 39: ABFV 208 UF VALVE
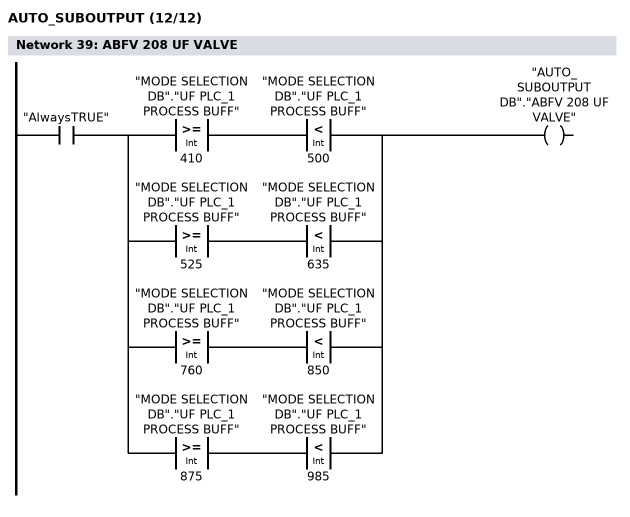
   RUNG wire#powerrail
      Contact( "AlwaysTRUE" )
      wire#w1
      { S7_Templates := "SrcType := Int" } GE_Contact(in1 := "MODE SELECTION DB"."UF PLC_1 PROCESS BUFF", in2 := 410)
      { S7_Templates := "SrcType := Int" } LT_Contact(in1 := "MODE SELECTION DB"."UF PLC_1 PROCESS BUFF", in2 := 500)
      wire#w2
      Coil( "AUTO_SUBOUTPUT DB"."ABFV 208 UF VALVE" )
   END_RUNG
   RUNG wire#w1
      { S7_Templates := "SrcType := Int" } GE_Contact(in1 := "MODE SELECTION DB"."UF PLC_1 PROCESS BUFF", in2 := 525)
      { S7_Templates := "SrcType := Int" } LT_Contact(in1 := "MODE SELECTION DB"."UF PLC_1 PROCESS BUFF", in2 := 635)
   END_RUNG wire#w2
   RUNG wire#w1
      { S7_Templates := "SrcType := Int" } GE_Contact(in1 := "MODE SELECTION DB"."UF PLC_1 PROCESS BUFF", in2 := 760)
      { S7_Templates := "SrcType := Int" } LT_Contact(in1 := "MODE SELECTION DB"."UF PLC_1 PROCESS BUFF", in2 := 850)
   END_RUNG wire#w2
   RUNG wire#w1
      { S7_Templates := "SrcType := Int" } GE_Contact(in1 := "MODE SELECTION DB"."UF PLC_1 PROCESS BUFF", in2 := 875)
      { S7_Templates := "SrcType := Int" } LT_Contact(in1 := "MODE SELECTION DB"."UF PLC_1 PROCESS BUFF", in2 := 985)
   END_RUNG wire#w2
   // the same network as SCL:
   "AUTO_SUBOUTPUT DB"."ABFV 208 UF VALVE" := "AlwaysTRUE" AND ((("MODE SELECTION DB"."UF PLC_1 PROCESS BUFF" >= 410) AND ("MODE SELECTION DB"."UF PLC_1 PROCESS BUFF" < 500)) OR (("MODE SELECTION DB"."UF PLC_1 PROCESS BUFF" >= 525) AND ("MODE SELECTION DB"."UF PLC_1 PROCESS BUFF" < 635)) OR (("MODE SELECTION DB"."UF PLC_1 PROCESS BUFF" >= 760) AND ("MODE SELECTION DB"."UF PLC_1 PROCESS BUFF" < 850)) OR (("MODE SELECTION DB"."UF PLC_1 PROCESS BUFF" >= 875) AND ("MODE SELECTION DB"."UF PLC_1 PROCESS BUFF" < 985)));
END_REGION
END_FUNCTION
